(* IEC 61131-3 sources: plc_simulator/services/codesys/POUs (part 10) *)

(* ---- TSK_FB_Analyze.st ---- *)
(* ============================================================
   TSK_FB_Analyze — Conflict analysis for task list
   ============================================================
   Ported from transporterTaskScheduler.js analyzeTaskConflicts()

   Three conflict checks, each stops at first hit:

   1. TASK_SEQUENCE: per-transporter queue order (preserves SWAP).
      Does the transporter have time to travel from prev.sink
      to next.lift?

   2. TRANSPORTER_COLLISION: different transporters — do their
      X-ranges and time-ranges overlap?

   3. CROSS_TRANSPORTER_HANDOFF: same batch, consecutive stages
      on different transporters — does the receiving transporter
      have time to reach the handoff station?

   NOTE: TASK_SEQUENCE iterates g_task[ti].Queue[] directly
   (not a merged sorted list) so SWAP ordering is preserved.

   Outputs:
     o_has_conflict — TRUE if conflict found
     o_conf_unit, o_conf_stage — which task is blocked
     o_blocked_unit, o_blocked_stage — which task blocks it
     o_deficit — how many seconds short
     o_conf_type — 1=TASK_SEQUENCE, 2=COLLISION, 3=HANDOFF
     checked_count — total tasks inspected
   ============================================================ *)

FUNCTION_BLOCK TSK_FB_Analyze
VAR_EXTERNAL CONSTANT
    MAX_Transporters    : INT;
    MAX_Units           : INT;
    MIN_StationIndex : INT;
    MAX_StationIndex   : INT;
END_VAR

VAR_EXTERNAL
  g_task    : ARRAY[1..MAX_Transporters] OF UDT_JC_TskQueueType;
  g_station : ARRAY[MIN_StationIndex..MAX_StationIndex] OF UDT_StationType;
  g_move    : ARRAY[1..MAX_Transporters] OF UDT_JC_MoveTimesType;
END_VAR
VAR_OUTPUT
  o_has_conflict  : BOOL;
  o_conf_type     : INT;     (* 1=TASK_SEQUENCE, 2=COLLISION, 3=HANDOFF *)
  o_conf_unit     : INT;     (* conflict task: unit *)
  o_conf_stage    : INT;     (* conflict task: stage *)
  o_conf_trans    : INT;     (* conflict task: transporter *)
  o_blocked_unit  : INT;     (* blocking task: unit *)
  o_blocked_stage : INT;     (* blocking task: stage *)
  o_deficit       : REAL;    (* seconds short *)
  checked_count   : INT;     (* tasks checked before conflict *)
END_VAR
VAR
  (* Loop variables *)
  ti       : INT;    (* transporter outer *)
  tj       : INT;    (* transporter inner *)
  qi       : INT;    (* queue index outer *)
  qj       : INT;    (* queue index inner *)
  (* TASK_SEQUENCE *)
  prev_sink : INT;
  next_lift : INT;
  travel_s  : REAL;
  gap_s     : REAL;
  deficit_s : REAL;
  (* TRANSPORTER_COLLISION: X range per task *)
  lift_x   : REAL;
  sink_x   : REAL;
  x1_min   : REAL;
  x1_max   : REAL;
  x2_min   : REAL;
  x2_max   : REAL;
  xo_start : REAL;
  xo_end   : REAL;
  to_start : LINT;
  to_end   : LINT;
  l_idx    : INT;
  s_idx    : INT;
  lift_x2  : REAL;
  sink_x2  : REAL;
  l_idx2   : INT;
  s_idx2   : INT;
  (* CROSS_TRANSPORTER_HANDOFF *)
  cur_unit    : INT;
  cur_stage   : INT;
  found_next  : BOOL;
  recv_prev_end  : LINT;
  recv_prev_sink : INT;
  has_recv_prev  : BOOL;
  rk       : INT;     (* receiver prev search *)
  recv_prev_unit : INT;    (* saved receiver prev task unit *)
  recv_prev_stg  : INT;    (* saved receiver prev task stage *)
  recv_travel    : REAL;
  recv_earliest  : LINT;
  handoff_deficit : REAL;
  (* Counter *)
  total_tasks : INT;
  DEFICIT_TOL : REAL := 1.0;
  tmp_move    : UDT_JC_MoveTimesType;  (* MATIEC cannot index arrays in FUNCTION args *)
END_VAR

o_has_conflict := FALSE;
o_conf_type    := 0;
o_deficit      := 0.0;
checked_count  := 0;

(* Count total tasks *)
total_tasks := 0;
FOR ti := 1 TO MAX_Transporters DO
  total_tasks := total_tasks + g_task[ti].Count;
END_FOR;
IF total_tasks = 0 THEN RETURN; END_IF;

(* ══════════════════════════════════════════════════════════════════════ *)
(* CHECK 1: TASK_SEQUENCE — per-transporter queue order (SWAP-safe)    *)
(* Iterates g_task[ti].Queue[] in queue order, NOT sorted by time.     *)
(* ══════════════════════════════════════════════════════════════════════ *)
FOR ti := 1 TO MAX_Transporters DO
  FOR qi := 1 TO g_task[ti].Count - 1 DO
    IF g_task[ti].Queue[qi].Unit > 0 AND g_task[ti].Queue[qi + 1].Unit > 0 THEN

      prev_sink := g_task[ti].Queue[qi].SinkStationTarget;
      next_lift := g_task[ti].Queue[qi + 1].LiftStationTarget;

      tmp_move := g_move[ti];
      travel_s := STC_CalcHorizontalTravel(i_from_stn := prev_sink, i_to_stn := next_lift, i_move := tmp_move);

      gap_s := LINT_TO_REAL(
        g_task[ti].Queue[qi + 1].StartTime - g_task[ti].Queue[qi].FinishTime
      );
      deficit_s := travel_s - gap_s;

      IF deficit_s > DEFICIT_TOL THEN
        o_has_conflict  := TRUE;
        o_conf_type     := 1;  (* TASK_SEQUENCE *)
        o_conf_unit     := g_task[ti].Queue[qi + 1].Unit;
        o_conf_stage    := g_task[ti].Queue[qi + 1].Stage;
        o_conf_trans    := ti;
        o_blocked_unit  := g_task[ti].Queue[qi].Unit;
        o_blocked_stage := g_task[ti].Queue[qi].Stage;
        o_deficit       := deficit_s;
        checked_count   := total_tasks;
        RETURN;
      END_IF;

    END_IF;
  END_FOR;
END_FOR;

(* ══════════════════════════════════════════════════════════════════════ *)
(* CHECK 2: CROSS_TRANSPORTER_HANDOFF                                  *)
(* Same batch, consecutive stages on different transporters.           *)
(* Does the receiving transporter have time to reach handoff station?  *)
(*                                                                      *)
(* JS checks HANDOFF before COLLISION (per-task loop order).           *)
(* Conflict targets the DELIVERING task (current transporter);         *)
(* resolver will delay the preceding stage so the batch waits longer   *)
(* on the delivering transporter's side.                               *)
(* ══════════════════════════════════════════════════════════════════════ *)
FOR ti := 1 TO MAX_Transporters DO
  FOR qi := 1 TO g_task[ti].Count DO
    cur_unit  := g_task[ti].Queue[qi].Unit;
    cur_stage := g_task[ti].Queue[qi].Stage;
    IF cur_unit > 0 THEN

      (* Find next stage of same batch in a different transporter *)
      found_next := FALSE;
      FOR tj := 1 TO MAX_Transporters DO
        IF tj <> ti AND NOT found_next THEN
          FOR qj := 1 TO g_task[tj].Count DO
            IF NOT found_next THEN
              IF g_task[tj].Queue[qj].Unit = cur_unit
                 AND g_task[tj].Queue[qj].Stage = cur_stage + 1 THEN
                found_next := TRUE;

                (* Found handoff pair: ti delivers to sink, tj picks up *)
                (* Find receiver's (tj) previous task — latest finish before next task start *)
                has_recv_prev := FALSE;
                recv_prev_end  := 0;
                recv_prev_sink := 0;
                recv_prev_unit := 0;
                recv_prev_stg  := 0;
                FOR rk := 1 TO g_task[tj].Count DO
                  IF rk <> qj THEN
                    IF g_task[tj].Queue[rk].FinishTime <= g_task[tj].Queue[qj].StartTime THEN
                      IF NOT has_recv_prev OR g_task[tj].Queue[rk].FinishTime > recv_prev_end THEN
                        has_recv_prev := TRUE;
                        recv_prev_end  := g_task[tj].Queue[rk].FinishTime;
                        recv_prev_sink := g_task[tj].Queue[rk].SinkStationTarget;
                        recv_prev_unit := g_task[tj].Queue[rk].Unit;
                        recv_prev_stg  := g_task[tj].Queue[rk].Stage;
                      END_IF;
                    END_IF;
                  END_IF;
                END_FOR;

                IF has_recv_prev THEN
                  (* Travel from receiver's prev sink to handoff station (= ti's current sink) *)
                  recv_travel := STC_CalcHorizontalTravel(
                    i_from_stn := recv_prev_sink,
                    i_to_stn   := g_task[ti].Queue[qi].SinkStationTarget,
                    i_move     := g_move[tj]
                  );
                  recv_earliest := recv_prev_end + REAL_TO_LINT(recv_travel);
                  handoff_deficit := LINT_TO_REAL(
                    recv_earliest - g_task[ti].Queue[qi].FinishTime
                  );

                  IF handoff_deficit > DEFICIT_TOL THEN
                    o_has_conflict  := TRUE;
                    o_conf_type     := 3;  (* CROSS_TRANSPORTER_HANDOFF *)
                    (* Conflict on delivering task *)
                    o_conf_unit     := g_task[ti].Queue[qi].Unit;
                    o_conf_stage    := g_task[ti].Queue[qi].Stage;
                    o_conf_trans    := ti;
                    (* Blocked by receiver's previous task *)
                    o_blocked_unit  := recv_prev_unit;
                    o_blocked_stage := recv_prev_stg;
                    o_deficit       := handoff_deficit;
                    checked_count   := total_tasks;
                    RETURN;
                  END_IF;
                END_IF;
                (* If no recv prev task, receiver is idle → no handoff conflict *)

              END_IF;
            END_IF;
          END_FOR;
        END_IF;
      END_FOR;

    END_IF;
  END_FOR;
END_FOR;

(* ══════════════════════════════════════════════════════════════════════ *)
(* CHECK 3: TRANSPORTER_COLLISION — X+time overlap, different trans.   *)
(* Compares every task pair across different transporters.              *)
(* JS: conf = later task (timeline), blocked = earlier task.           *)
(* ══════════════════════════════════════════════════════════════════════ *)
FOR ti := 1 TO MAX_Transporters DO
  FOR qi := 1 TO g_task[ti].Count DO
    IF g_task[ti].Queue[qi].Unit > 0 THEN

      (* X range for task A *)
      l_idx := g_task[ti].Queue[qi].LiftStationTarget - 100;
      s_idx := g_task[ti].Queue[qi].SinkStationTarget - 100;
      IF l_idx >= 1 AND l_idx <= 30 THEN
        lift_x := DINT_TO_REAL(g_station[g_task[ti].Queue[qi].LiftStationTarget].XPosition);
      ELSE
        lift_x := 0.0;
      END_IF;
      IF s_idx >= 1 AND s_idx <= 30 THEN
        sink_x := DINT_TO_REAL(g_station[g_task[ti].Queue[qi].SinkStationTarget].XPosition);
      ELSE
        sink_x := 0.0;
      END_IF;
      IF lift_x < sink_x THEN
        x1_min := lift_x;
        x1_max := sink_x;
      ELSE
        x1_min := sink_x;
        x1_max := lift_x;
      END_IF;

      FOR tj := ti + 1 TO MAX_Transporters DO
        FOR qj := 1 TO g_task[tj].Count DO
          IF g_task[tj].Queue[qj].Unit > 0 THEN

            (* X range for task B *)
            l_idx2 := g_task[tj].Queue[qj].LiftStationTarget - 100;
            s_idx2 := g_task[tj].Queue[qj].SinkStationTarget - 100;
            IF l_idx2 >= 1 AND l_idx2 <= 30 THEN
              lift_x2 := DINT_TO_REAL(g_station[g_task[tj].Queue[qj].LiftStationTarget].XPosition);
            ELSE
              lift_x2 := 0.0;
            END_IF;
            IF s_idx2 >= 1 AND s_idx2 <= 30 THEN
              sink_x2 := DINT_TO_REAL(g_station[g_task[tj].Queue[qj].SinkStationTarget].XPosition);
            ELSE
              sink_x2 := 0.0;
            END_IF;
            IF lift_x2 < sink_x2 THEN
              x2_min := lift_x2;
              x2_max := sink_x2;
            ELSE
              x2_min := sink_x2;
              x2_max := lift_x2;
            END_IF;

            (* X overlap *)
            xo_start := x1_min;
            IF x2_min > xo_start THEN xo_start := x2_min; END_IF;
            xo_end := x1_max;
            IF x2_max < xo_end THEN xo_end := x2_max; END_IF;

            IF xo_start < xo_end THEN
              (* Time overlap *)
              to_start := g_task[ti].Queue[qi].StartTime;
              IF g_task[tj].Queue[qj].StartTime > to_start THEN
                to_start := g_task[tj].Queue[qj].StartTime;
              END_IF;
              to_end := g_task[ti].Queue[qi].FinishTime;
              IF g_task[tj].Queue[qj].FinishTime < to_end THEN
                to_end := g_task[tj].Queue[qj].FinishTime;
              END_IF;

              IF to_start < to_end THEN
                deficit_s := LINT_TO_REAL(to_end - to_start) + 2.0;
                o_has_conflict  := TRUE;
                o_conf_type     := 2;  (* TRANSPORTER_COLLISION *)
                (* Assign conf = later task (timeline), blocked = earlier task — matches JS *)
                IF g_task[ti].Queue[qi].StartTime <= g_task[tj].Queue[qj].StartTime THEN
                  o_conf_unit     := g_task[tj].Queue[qj].Unit;
                  o_conf_stage    := g_task[tj].Queue[qj].Stage;
                  o_conf_trans    := tj;
                  o_blocked_unit  := g_task[ti].Queue[qi].Unit;
                  o_blocked_stage := g_task[ti].Queue[qi].Stage;
                ELSE
                  o_conf_unit     := g_task[ti].Queue[qi].Unit;
                  o_conf_stage    := g_task[ti].Queue[qi].Stage;
                  o_conf_trans    := ti;
                  o_blocked_unit  := g_task[tj].Queue[qj].Unit;
                  o_blocked_stage := g_task[tj].Queue[qj].Stage;
                END_IF;
                o_deficit       := deficit_s;
                checked_count   := total_tasks;
                RETURN;
              END_IF;
            END_IF;

          END_IF;
        END_FOR;
      END_FOR;

    END_IF;
  END_FOR;
END_FOR;

(* No conflict found *)
checked_count := total_tasks;

END_FUNCTION_BLOCK

(* ---- TSK_FB_CalcSchedule.st ---- *)
(* ============================================================
   TSK_FB_CalcSchedule — Calculate batch schedule for one unit
   ============================================================
   Ported from transporterTaskScheduler.js calculateBatchSchedule()

   Calculates schedule timeline for one unit/batch:
   - Reads treatment program stages
   - Calculates transfer times from g_move
   - Writes entry/exit times to g_schedule[unit]

   Parallel stations: picks first available (stations[1] default).
   Transfer time: lift + travel + sink from g_move precomputed table.

   Called once per batch per scheduler cycle.
   ============================================================ *)

FUNCTION_BLOCK TSK_FB_CalcSchedule
VAR_INPUT
  i_unit     : INT;     (* unit index 1..10 *)
  i_trans    : INT;     (* transporter index 1..3 for move times *)
  i_time_s   : LINT;    (* current absolute time (s), unix seconds *)
END_VAR
VAR_EXTERNAL CONSTANT
    MIN_StationIndex : INT;
    MAX_StationIndex   : INT;
    MAX_Units           : INT;
    MAX_Transporters    : INT;
END_VAR
VAR_EXTERNAL
  g_batch  : ARRAY[1..MAX_Units] OF UDT_BatchType;
  g_program : ARRAY[1..MAX_Units] OF UDT_TreatmentProgramType;
  g_unit    : ARRAY[1..MAX_Units] OF UDT_UnitType;
  g_station : ARRAY[MIN_StationIndex..MAX_StationIndex] OF UDT_StationType;
  g_station_loc : ARRAY[1..MAX_StationIndex] OF UDT_UnitLocation;
  g_schedule : ARRAY[1..MAX_Units] OF UDT_JC_TskScheduleType;
  g_station_count : INT;
  g_move    : ARRAY[1..MAX_Transporters] OF UDT_JC_MoveTimesType;
  g_cfg     : ARRAY[1..MAX_Transporters] OF UDT_TransporterType;
  g_transporter : ARRAY[1..MAX_Transporters] OF UDT_TransporterStatusType;
END_VAR
VAR
  stg         : INT;      (* loop: stage index *)
  stn_num    : INT;      (* target station number *)
  prev_stn   : INT;      (* previous station number *)
  cur_stage  : INT;      (* batch current stage *)
  location   : INT;      (* unit location *)
  start_st   : INT;      (* first stage to calculate *)
  entry_t    : LINT;     (* entry time for stage, absolute *)
  exit_t     : LINT;     (* exit time for stage, absolute *)
  xfer_t     : REAL;     (* transfer time *)
  calc_s     : REAL;     (* calc_time in seconds *)
  min_s      : REAL;     (* min_time in seconds *)
  max_s      : REAL;     (* max_time in seconds *)
  is_on_stn  : BOOL;     (* TRUE if unit is on a station *)
  is_first   : BOOL;     (* TRUE for first stage in loop *)
  remain_s   : REAL;     (* remaining time on current station *)
  elapsed_s  : REAL;     (* elapsed time on current station *)
  out_count  : INT;      (* output stage counter *)
  p          : INT;      (* parallel station loop index *)
  chosen_stn : INT;      (* chosen parallel station *)
  tmp_move   : UDT_JC_MoveTimesType;  (* MATIEC cannot index arrays in FUNCTION args *)
  (* ── Parallel station selection (schedule-aware + idle-since) ── *)
  cand_arr         : ARRAY[1..5] OF INT;
  cand_cnt         : INT;
  sched_occupied   : ARRAY[1..5] OF BOOL;
  phys_occupied    : ARRAY[1..5] OF BOOL;
  best_change_time : LINT;
  my_entry         : LINT;
  my_exit          : LINT;
  ov_start         : LINT;
  ov_end           : LINT;
  uj               : INT;
  sj               : INT;
  saved_entry_t    : LINT;  (* previous cycle's first-stage EntryTime for on-transporter clamp *)
END_VAR

(* -- Validate inputs -- *)
IF i_unit < 1 OR i_unit > MAX_Units THEN RETURN; END_IF;
IF i_trans < 1 OR i_trans > MAX_Transporters THEN RETURN; END_IF;

(* -- Read batch and unit data -- *)
cur_stage := g_batch[i_unit].CurStage;
location  := g_unit[i_unit].location;
is_on_stn := location >= 100;
out_count := 0;

(* -- Save previous first-stage entry time before clearing -- *)
(* When unit is on transporter, we preserve the previously calculated
   entry time as long as it is still in the future (= transporter on schedule).
   If it has passed, we clamp to now (= transporter is late). *)
saved_entry_t := 0;
IF NOT is_on_stn AND g_schedule[i_unit].StageCount > 0 THEN
  saved_entry_t := g_schedule[i_unit].Stages[1].EntryTime;
END_IF;

(* -- Clear old schedule -- *)
FOR stg := 1 TO 30 DO
  g_schedule[i_unit].Stages[stg].station := 0;
  g_schedule[i_unit].Stages[stg].ProgramStage := 0;
  g_schedule[i_unit].Stages[stg].EntryTime := 0;
  g_schedule[i_unit].Stages[stg].ExitTime := 0;
  g_schedule[i_unit].Stages[stg].MinTime := 0;
  g_schedule[i_unit].Stages[stg].CalcTime := 0;
  g_schedule[i_unit].Stages[stg].MaxTime := 0;
  g_schedule[i_unit].Stages[stg].TransferTime := 0;
END_FOR;

(* -- Determine start stage -- *)
(* Waiting batch (state = NOT_PROCESSED): treat as stage 0 *)
IF g_batch[i_unit].State = 0 THEN
  cur_stage := 0;
END_IF;

(* If on transporter, start from next stage; if on station, from current *)
IF is_on_stn THEN
  start_st := cur_stage;
ELSE
  start_st := cur_stage + 1;
END_IF;

(* Force minimum stage 1 *)
IF start_st < 1 THEN
  start_st := 1;
END_IF;

(* -- Previous station (where transfer starts from) -- *)
IF is_on_stn THEN
  prev_stn := location;
ELSIF cur_stage >= 1 AND cur_stage <= 30 THEN
  (* On transporter: use previous stage station *)
  prev_stn := g_program[i_unit].Steps[cur_stage].Stations[0];
ELSE
  prev_stn := 0;
END_IF;

(* -- prevExitTime: when next stage can begin -- *)
exit_t := i_time_s;

is_first := TRUE;

(* -- Prepend current location when unit needs pre-positioning -- *)
(* If unit is on a station that is NOT the first treatment station,
   insert it as schedule entry 0 (0 treatment time) so that
   CreateTasks generates a move-to-first-station task. *)
IF is_on_stn AND start_st >= 1 THEN
  stn_num := 0;
  FOR p := 0 TO 4 DO
    IF g_program[i_unit].Steps[start_st].Stations[p] = location THEN
      stn_num := location;  (* flag: already on first treatment station *)
    END_IF;
  END_FOR;
  IF stn_num = 0 THEN
    out_count := out_count + 1;
    g_schedule[i_unit].Stages[out_count].station       := location;
    g_schedule[i_unit].Stages[out_count].ProgramStage := 0;  (* pre-position entry, not a program stage *)
    g_schedule[i_unit].Stages[out_count].EntryTime    := exit_t;
    g_schedule[i_unit].Stages[out_count].TransferTime := 0;

    (* ── Stage 0 times from batch data — JS: stage0 prepend uses batch.calc/min/max ──
       CurStage=0 means just activated: use batch CalTime (= remaining wait time)
       Otherwise (mid-process repositioning): zero duration *)
    IF g_batch[i_unit].CurStage = 0 AND g_batch[i_unit].CalTime > 0 THEN
      (* JS: remainingSec = max(1, calcTimeS - elapsed) *)
      IF g_batch[i_unit].StartTime > 0 AND g_batch[i_unit].StartTime < i_time_s THEN
        elapsed_s := LINT_TO_REAL(i_time_s - g_batch[i_unit].StartTime);
      ELSE
        elapsed_s := 0.0;
      END_IF;
      remain_s := DINT_TO_REAL(g_batch[i_unit].CalTime) - elapsed_s;
      IF remain_s < 1.0 THEN remain_s := 1.0; END_IF;
      exit_t := i_time_s + REAL_TO_LINT(remain_s);
      g_schedule[i_unit].Stages[out_count].ExitTime  := exit_t;
      g_schedule[i_unit].Stages[out_count].CalcTime  := REAL_TO_DINT(remain_s);
      g_schedule[i_unit].Stages[out_count].MinTime   := g_batch[i_unit].MinTime;
      g_schedule[i_unit].Stages[out_count].MaxTime   := g_batch[i_unit].MaxTime;
    ELSE
      g_schedule[i_unit].Stages[out_count].ExitTime  := exit_t;
      g_schedule[i_unit].Stages[out_count].CalcTime  := 0;
      g_schedule[i_unit].Stages[out_count].MinTime   := 0;
      g_schedule[i_unit].Stages[out_count].MaxTime   := 0;
    END_IF;

    is_first := FALSE;
  END_IF;
END_IF;

(* ============================================================
   MAIN LOOP: Calculate schedule for each program stage
   ============================================================ *)
FOR stg := start_st TO g_program[i_unit].StepCount DO

  (* Check if stage has valid stations — parallel selection *)
  cand_cnt := 0;
  FOR p := 0 TO 4 DO
    IF g_program[i_unit].Steps[stg].Stations[p] > 0 THEN
      cand_cnt := cand_cnt + 1;
      cand_arr[cand_cnt] := g_program[i_unit].Steps[stg].Stations[p];
      sched_occupied[cand_cnt] := FALSE;
      phys_occupied[cand_cnt] := FALSE;
    END_IF;
  END_FOR;

  (* No station means end of program *)
  IF cand_cnt = 0 THEN
    EXIT;
  END_IF;

  IF cand_cnt = 1 THEN
    chosen_stn := cand_arr[1];
  ELSE
    (* Read treatment times early — needed for time window estimate *)
    calc_s := DINT_TO_REAL(g_program[i_unit].Steps[stg].CalTime);

    (* Estimate this stage's time window *)
    tmp_move := g_move[i_trans];
    xfer_t := STC_CalcTransferTime(
      i_from_stn            := prev_stn,
      i_to_stn              := cand_arr[1],
      i_move                := tmp_move,
      i_from_dropping_x10   := g_station[prev_stn].DrippingTime,
      i_to_device_delay_x10 := g_station[cand_arr[1]].DeviceDelay,
      i_drip_tray_delay_x10 := g_cfg[i_trans].DripTrayDelay
    );
    my_entry := exit_t + REAL_TO_LINT(xfer_t);
    my_exit  := my_entry + REAL_TO_LINT(calc_s);

    (* Check schedule overlap + physical occupation for each candidate *)
    FOR p := 1 TO cand_cnt DO
      FOR uj := 1 TO MAX_Units DO
        IF uj <> i_unit AND g_schedule[uj].StageCount > 0 THEN
          FOR sj := 1 TO g_schedule[uj].StageCount DO
            IF g_schedule[uj].Stages[sj].station = cand_arr[p] THEN
              ov_start := my_entry;
              IF g_schedule[uj].Stages[sj].EntryTime > ov_start THEN
                ov_start := g_schedule[uj].Stages[sj].EntryTime;
              END_IF;
              ov_end := my_exit;
              IF g_schedule[uj].Stages[sj].ExitTime < ov_end THEN
                ov_end := g_schedule[uj].Stages[sj].ExitTime;
              END_IF;
              IF ov_end > ov_start THEN
                sched_occupied[p] := TRUE;
              END_IF;
            END_IF;
          END_FOR;
        END_IF;
      END_FOR;

      (* Physical occupation *)
      FOR uj := 1 TO MAX_Units DO
        IF g_unit[uj].location = cand_arr[p] AND g_unit[uj].Status = 1 THEN
          phys_occupied[p] := TRUE;
        END_IF;
      END_FOR;
    END_FOR;

    (* Select best free station: longest idle = smallest change_time *)
    chosen_stn := 0;
    best_change_time := LINT#9999999999;
    FOR p := 1 TO cand_cnt DO
      IF NOT sched_occupied[p] AND NOT phys_occupied[p] THEN
        IF cand_arr[p] >= MIN_StationIndex AND cand_arr[p] <= MAX_StationIndex THEN
          IF g_station_loc[cand_arr[p]].ChangeTime < best_change_time THEN
            best_change_time := g_station_loc[cand_arr[p]].ChangeTime;
            chosen_stn := cand_arr[p];
          END_IF;
        END_IF;
      END_IF;
    END_FOR;

    (* Fallback: schedule-free only *)
    IF chosen_stn = 0 THEN
      FOR p := 1 TO cand_cnt DO
        IF NOT sched_occupied[p] AND chosen_stn = 0 THEN
          chosen_stn := cand_arr[p];
        END_IF;
      END_FOR;
    END_IF;

    (* Ultimate fallback: first candidate *)
    IF chosen_stn = 0 THEN
      chosen_stn := cand_arr[1];
    END_IF;
  END_IF;

  stn_num := chosen_stn;

  (* Read treatment times from program *)
  calc_s := DINT_TO_REAL(g_program[i_unit].Steps[stg].CalTime);
  min_s  := DINT_TO_REAL(g_program[i_unit].Steps[stg].MinTime);
  max_s  := DINT_TO_REAL(g_program[i_unit].Steps[stg].MaxTime);

  (* -- Calculate transfer time from prev_stn to stn_num -- *)
  (* Cross-transfer check: if prev_stn has Crosstransport and different Y line
     → use ChangeStation as effective source for transfer time calc
     JS: calculateTransferTimeWithCrossCheck *)
  tmp_move := g_move[i_trans];
  (* ST does NOT short-circuit AND — bounds must be checked in separate IF
     before any g_station[prev_stn] or g_station[stn_num] access *)
  IF prev_stn >= MIN_StationIndex AND prev_stn <= MAX_StationIndex
     AND stn_num >= MIN_StationIndex AND stn_num <= MAX_StationIndex THEN
    IF g_station[prev_stn].Crosstransport > 0
       AND g_station[prev_stn].ChangeStation > 0
       AND g_station[prev_stn].YPosition <> g_station[stn_num].YPosition THEN
      (* Cross-transfer: belt time + transfer from ChangeStation to sink *)
      xfer_t := INT_TO_REAL(g_station[prev_stn].CrossTransportTime)
              + STC_CalcTransferTime(
                  i_from_stn            := g_station[prev_stn].ChangeStation,
                  i_to_stn              := stn_num,
                  i_move                := tmp_move,
                  i_from_dropping_x10   := g_station[g_station[prev_stn].ChangeStation].DrippingTime,
                  i_to_device_delay_x10 := g_station[stn_num].DeviceDelay,
                  i_drip_tray_delay_x10 := g_cfg[i_trans].DripTrayDelay
                );
    ELSE
      xfer_t := STC_CalcTransferTime(
        i_from_stn            := prev_stn,
        i_to_stn              := stn_num,
        i_move                := tmp_move,
        i_from_dropping_x10   := g_station[prev_stn].DrippingTime,
        i_to_device_delay_x10 := g_station[stn_num].DeviceDelay,
        i_drip_tray_delay_x10 := g_cfg[i_trans].DripTrayDelay
      );
    END_IF;
  ELSE
    (* Out-of-range station index — use safe fallback *)
    xfer_t := 60.0;
  END_IF;

  (* -- Calculate entry and exit times -- *)
  IF is_first AND is_on_stn AND stg = cur_stage THEN
    (* Batch is currently at this station *)
    entry_t := i_time_s;
    (* Remaining time: use g_batch[].CalTime (resolver-modified)
       JS: remainingTimeS = max(1, batch.calc_time_s - elapsed) *)
    IF g_batch[i_unit].StartTime > 0 THEN
      elapsed_s := LINT_TO_REAL(i_time_s - g_batch[i_unit].StartTime);
    ELSE
      elapsed_s := 0.0;
    END_IF;
    remain_s := DINT_TO_REAL(g_batch[i_unit].CalTime) - elapsed_s;
    IF remain_s < 1.0 THEN remain_s := 1.0; END_IF;
    exit_t := i_time_s + REAL_TO_LINT(remain_s);
  ELSIF is_first AND NOT is_on_stn THEN
    (* Batch is on transporter — use saved entry time from previous cycle.
       If transporter is on schedule (saved > now), keep it stable.
       If transporter is late (saved <= now), clamp to now. *)
    IF saved_entry_t > i_time_s THEN
      entry_t := saved_entry_t;  (* on schedule — keep stable *)
    ELSE
      entry_t := i_time_s;       (* late or first cycle — clamp to now *)
    END_IF;
    exit_t  := entry_t + REAL_TO_LINT(calc_s);
  ELSE
    (* Normal stage: entry = prev exit + transfer *)
    entry_t := exit_t + REAL_TO_LINT(xfer_t);
    exit_t  := entry_t + REAL_TO_LINT(calc_s);
  END_IF;

  (* -- Write to schedule -- *)
  out_count := out_count + 1;
  IF out_count <= 30 THEN
    g_schedule[i_unit].Stages[out_count].station       := stn_num;
    g_schedule[i_unit].Stages[out_count].ProgramStage := stg;  (* program stage number (1..N) *)
    g_schedule[i_unit].Stages[out_count].EntryTime    := entry_t;
    g_schedule[i_unit].Stages[out_count].ExitTime     := exit_t;
    g_schedule[i_unit].Stages[out_count].MinTime      := REAL_TO_DINT(min_s);
    g_schedule[i_unit].Stages[out_count].CalcTime     := REAL_TO_DINT(calc_s);
    g_schedule[i_unit].Stages[out_count].MaxTime      := REAL_TO_DINT(max_s);
    g_schedule[i_unit].Stages[out_count].TransferTime := REAL_TO_DINT(xfer_t);
  END_IF;

  (* -- Update for next iteration -- *)
  prev_stn := stn_num;
  is_first := FALSE;

END_FOR;

g_schedule[i_unit].StageCount := out_count;

END_FUNCTION_BLOCK

(* ---- TSK_FB_CreateTasks.st ---- *)
(* ============================================================
   TSK_FB_CreateTasks — Build task list from schedule
   ============================================================
   Ported from transporterTaskScheduler.js createTaskListFromSchedule()

   For each consecutive stage pair in g_schedule[unit]:
     - Lift station = current stage station
     - Sink station = next stage station
     - Assigns transporter from task_area match in g_cfg
     - Skips already completed stages (stage < batch.CurStage)
   Appends tasks to g_task[transporter].Queue.

   Called once per batch per scheduler cycle.
   ============================================================ *)

FUNCTION_BLOCK TSK_FB_CreateTasks
VAR_INPUT
  i_unit : INT;   (* unit index 1..10 *)
END_VAR
VAR_EXTERNAL CONSTANT
    MAX_Transporters : INT;
    MAX_Units        : INT;
    MAX_TASK_QUEUE   : INT;
    MIN_StationIndex : INT;
    MAX_StationIndex : INT;
END_VAR

VAR_EXTERNAL
  g_batch  : ARRAY[1..MAX_Units] OF UDT_BatchType;
  g_schedule : ARRAY[1..MAX_Units] OF UDT_JC_TskScheduleType;
  g_task    : ARRAY[1..MAX_Transporters] OF UDT_JC_TskQueueType;
  g_cfg    : ARRAY[1..MAX_Transporters] OF UDT_TransporterType;
  g_station : ARRAY[MIN_StationIndex..MAX_StationIndex] OF UDT_StationType;
END_VAR
VAR
  si         : INT;     (* schedule stage index *)
  sc         : INT;     (* stage count *)
  lift_stn   : INT;     (* lift station *)
  sink_stn   : INT;     (* sink station *)
  tid        : INT;     (* transporter id found *)
  qi         : INT;     (* queue write index *)
  fb_find    : STC_FindTransporter;  (* transporter lookup *)
  (* Cross-transfer detection — JS: isCrossTransporterOp + findCrossTransporterEndStation *)
  eff_lift_stn : INT;   (* effective lift station after cross-transfer check *)
END_VAR

IF i_unit < 1 OR i_unit > MAX_Units THEN RETURN; END_IF;

sc := g_schedule[i_unit].StageCount;
IF sc < 2 THEN RETURN; END_IF;

(* CalcSchedule already builds a schedule starting from the batch's
   current stage (and prepends the unit's current location when needed).
   No skip logic needed here — every consecutive pair is a valid task. *)

(* Loop through consecutive stage pairs *)
FOR si := 1 TO sc - 1 DO
  lift_stn := g_schedule[i_unit].Stages[si].station;
  sink_stn := g_schedule[i_unit].Stages[si + 1].station;

  IF lift_stn > 0 AND sink_stn > 0 THEN
    (* -- Cross-transfer detection -- *)
    (* JS: if station.operation === 10 && lift.y_position !== sink.y_position
       → use ChangeStation as effective lift (belt other end, same line as sink) *)
    eff_lift_stn := lift_stn;
    IF lift_stn >= MIN_StationIndex AND lift_stn <= MAX_StationIndex
       AND sink_stn >= MIN_StationIndex AND sink_stn <= MAX_StationIndex THEN
      IF g_station[lift_stn].Crosstransport > 0
         AND g_station[lift_stn].ChangeStation > 0
         AND g_station[lift_stn].YPosition <> g_station[sink_stn].YPosition THEN
        eff_lift_stn := g_station[lift_stn].ChangeStation;
      END_IF;
    END_IF;

    (* -- Find transporter via task_area matching (with scoring) -- *)
    fb_find(i_lift_stn := eff_lift_stn, i_sink_stn := sink_stn);
    tid := fb_find.o_trans;

    (* -- Append task to transporter queue -- *)
    IF tid >= 1 AND tid <= 3 THEN
      qi := g_task[tid].Count + 1;
      IF qi <= MAX_TASK_QUEUE THEN
        g_task[tid].Queue[qi].Unit         := i_unit;
        g_task[tid].Queue[qi].Stage        := g_schedule[i_unit].Stages[si].ProgramStage;  (* program stage — direct index to g_program.Steps[] *)
        g_task[tid].Queue[qi].LiftStationTarget := eff_lift_stn;
        g_task[tid].Queue[qi].SinkStationTarget := sink_stn;
        g_task[tid].Queue[qi].StartTime   := g_schedule[i_unit].Stages[si].ExitTime;
        g_task[tid].Queue[qi].FinishTime  := g_schedule[i_unit].Stages[si + 1].EntryTime;
        g_task[tid].Queue[qi].CalcTime    := g_schedule[i_unit].Stages[si].CalcTime;
        g_task[tid].Queue[qi].MinTime     := g_schedule[i_unit].Stages[si].MinTime;
        g_task[tid].Queue[qi].MaxTime     := g_schedule[i_unit].Stages[si].MaxTime;
        g_task[tid].Count := qi;
      END_IF;
    END_IF;
  END_IF;
END_FOR;

END_FUNCTION_BLOCK

(* ---- TSK_FB_NoTreatment.st ---- *)
(* ============================================================
   TSK_FB_NoTreatment — Create no-treatment transfer tasks
   ============================================================
   Scans units that have a target (TO_LOADING, TO_UNLOAD,
   TO_BUFFER, TO_AVOID, etc.) and creates transfer tasks using
   the g_ntt destination table (per target, per transporter).

   Destination lookup:
     1. Search primary stations (g_ntt[trans].Target[tgt].Stations)
     2. If all occupied → search fallback stations
     3. First free station wins

   Conditions for creating a task:
     - Unit has target <> TO_NONE
     - TO_PROCESS handled only when batch state = NOT_PROCESSED
       (routes to loaded-buffer via NTT index 7)
     - Unit is on a station (location >= 100)
     - Covering transporter is idle (phase = 0, active)
     - A free destination station exists in g_ntt
     - Destination station MUST be actually free (no unit present)
     - No overlap conflict with OTHER transporters that share the
       destination area (mirrors JS _hasOverlapConflict):
       * If another transporter also covers dest_stn and is actively
         moving (Phase 1-4) with its task in the shared zone → skip
       * If another transporter has queued tasks that overlap in time
         AND operate in cov_t's task area → skip
   ============================================================ *)

FUNCTION_BLOCK TSK_FB_NoTreatment
VAR_INPUT
  i_time_s : LINT;   (* current absolute time (s), unix seconds *)
END_VAR
VAR_EXTERNAL CONSTANT
    MAX_Transporters    : INT;
    MAX_STATIONS_PER_STEP       : INT;
    MIN_StationIndex : INT;
    MAX_StationIndex   : INT;
    MAX_Units           : INT;
    MAX_TASK_QUEUE      : INT;
END_VAR

VAR_EXTERNAL
  g_unit        : ARRAY[1..MAX_Units] OF UDT_UnitType;
  g_batch       : ARRAY[1..MAX_Units] OF UDT_BatchType;
  g_ntt         : ARRAY[1..MAX_Transporters] OF UDT_JC_NttTransporterType;
  g_transporter : ARRAY[1..MAX_Transporters] OF UDT_TransporterStatusType;
  g_station     : ARRAY[MIN_StationIndex..MAX_StationIndex] OF UDT_StationType;
  g_station_loc : ARRAY[1..MAX_StationIndex] OF UDT_UnitLocation;
  g_cfg         : ARRAY[1..MAX_Transporters] OF UDT_TransporterType;
  g_task        : ARRAY[1..MAX_Transporters] OF UDT_JC_TskQueueType;
  g_move        : ARRAY[1..MAX_Transporters] OF UDT_JC_MoveTimesType;
END_VAR
VAR
  ui       : INT;     (* unit loop *)
  qi       : INT;     (* queue index *)
  loc      : INT;     (* unit location station *)
  tgt      : INT;     (* unit target *)
  cov_t    : INT;     (* transporter loop *)
  ai       : INT;     (* task_area loop *)
  covers   : BOOL;    (* transporter covers this station *)
  done     : BOOL;    (* task created for this unit *)
  dest     : UDT_JC_NttDestType;  (* destination descriptor for this target+transporter *)
  ntt_idx  : INT;     (* resolved NTT index (maps TO_BUFFER to 6/7/8 based on batch) *)
  (* Location classification *)
  on_primary  : BOOL;  (* unit is already on a primary station *)
  on_fallback : BOOL;  (* unit is on a fallback station *)
  primary_free : BOOL; (* at least one primary station is free *)
  (* Destination search *)
  dest_stn : INT;     (* destination station *)
  si       : INT;     (* station loop *)
  station_idx      : INT;     (* candidate station *)
  stn_free : BOOL;
  uj       : INT;     (* inner unit loop for free check *)
  (* Duplicate check *)
  ti       : INT;     (* inner transporter loop *)
  already  : BOOL;    (* unit already queued or being transported *)
  qi2      : INT;     (* queue scan index *)
  (* Timing *)
  xfer_s   : REAL;    (* total transfer time *)
  task_start : LINT;
  task_end   : LINT;
  (* Idle-slot overlap check *)
  has_overlap    : BOOL;
  ntt_start      : LINT;
  ntt_end        : LINT;
  ov_s           : LINT;
  ov_e           : LINT;
  margin_travel  : REAL;
  slot_start     : LINT;   (* idle slot bounds *)
  tmp_move       : UDT_JC_MoveTimesType;  (* MATIEC cannot index arrays in FUNCTION args *)
  slot_end       : LINT;
  earliest_start : LINT;   (* earliest NTT start considering travel *)
  latest_end     : LINT;   (* latest NTT end considering travel *)
  travel_to_lift : REAL;
  travel_from_sink : REAL;
  ntt_duration   : LINT;
  qi3            : INT;   (* queue loop for idle-slot calc *)
  slot_ok        : BOOL;
  sh             : INT;   (* shift loop for insert-at-first *)
  (* Multi-transporter shared-area idle check *)
  ot             : INT;   (* other transporter loop *)
  oq             : INT;   (* other transporter queue loop *)
  overlap_conflict : BOOL;
  dest_x         : DINT;  (* dest_stn X position mm *)
  avoid_dist     : DINT;  (* cov_t avoid distance mm *)
  cov_min_x      : DINT;  (* cov_t drive limit min mm *)
  cov_max_x      : DINT;  (* cov_t drive limit max mm *)
  ot_min_x       : DINT;  (* other transporter drive limit min mm *)
  ot_max_x       : DINT;  (* other transporter drive limit max mm *)
  zone_min_x     : DINT;  (* shared overlap zone min mm *)
  zone_max_x     : DINT;  (* shared overlap zone max mm *)
  danger_min     : DINT;  (* zone_min - avoid_dist *)
  danger_max     : DINT;  (* zone_max + avoid_dist *)
  (* Shared-area timing: NTT split into own-area + shared-area portions *)
  loc_idx        : INT;   (* from_stn index = loc - 100 *)
  loc_x          : DINT;  (* lift station X position mm *)
  phase2_s       : REAL;  (* Phase 2 duration: lift + drip + tray (own area time) *)
  shared_entry   : LINT;  (* time when NTT enters shared area *)
  shared_time    : REAL;  (* duration NTT is on shared area *)
  ot_idle_ok     : BOOL;  (* other transporter has sufficient idle window *)
  ot_idle_start  : LINT;  (* other transporter idle window start *)
  ot_idle_end    : LINT;  (* other transporter idle window end *)
END_VAR

FOR ui := 1 TO MAX_Units DO
  tgt := g_unit[ui].Target;
  loc := g_unit[ui].location;

  (* Skip: no target, not on station.
     TO_PROCESS(3) is only handled here when batch state = NOT_PROCESSED
     (loaded unit waiting for processing → route to loaded-buffer). *)
  IF tgt >= 1 AND tgt <= 5 AND loc >= 100 THEN

    (* TO_PROCESS with batch already IN_PROCESS or later → skip (handled by schedule) *)
    IF tgt = 3 AND (g_batch[ui].BatchCode = 0 OR g_batch[ui].State <> 0) THEN
      CONTINUE;
    END_IF;

    (* Skip if unit already has a pending task in any queue or is being transported *)
    already := FALSE;
    FOR ti := 1 TO MAX_Transporters DO
      IF NOT already THEN
        (* Being transported right now? *)
        IF g_transporter[ti].Phase > 0 AND g_station_loc[ti].UnitId = ui THEN
          already := TRUE;
        END_IF;
        (* In any task queue? *)
        FOR qi2 := 1 TO g_task[ti].Count DO
          IF NOT already THEN
            IF g_task[ti].Queue[qi2].Unit = ui THEN
              already := TRUE;
            END_IF;
          END_IF;
        END_FOR;
      END_IF;
    END_FOR;

    IF NOT already THEN

    (* Try each transporter — not just the first covering one *)
    done := FALSE;
    FOR cov_t := 1 TO MAX_Transporters DO
      IF NOT done THEN

      (* Check coverage: transporter task_area covers this station *)
      covers := FALSE;
      FOR ai := 1 TO 4 DO
        IF NOT covers THEN
          IF g_cfg[cov_t].TaskArea[ai].MinLift > 0 OR g_cfg[cov_t].TaskArea[ai].MaxLift > 0 THEN
            IF loc >= g_cfg[cov_t].TaskArea[ai].MinLift AND loc <= g_cfg[cov_t].TaskArea[ai].MaxLift THEN
              covers := TRUE;
            END_IF;
          END_IF;
        END_IF;
      END_FOR;

      IF covers AND g_transporter[cov_t].IsActive
         AND (g_transporter[cov_t].Phase = 0 OR tgt = 5) THEN

        (* ── Resolve NTT index ── *)
        (* TO_BUFFER(2) maps to 6/7/8 depending on batch state *)
        (* TO_PROCESS(3) with NOT_PROCESSED batch → loaded buffer (7) *)
        IF tgt = 2 THEN
          IF g_batch[ui].BatchCode = 0 THEN
            ntt_idx := 6;  (* empty buffer — no batch *)
          ELSIF g_batch[ui].State = 2 THEN
            ntt_idx := 8;  (* processed buffer — batch PROCESSED *)
          ELSE
            ntt_idx := 7;  (* loaded buffer — batch NOT_PROCESSED or IN_PROCESS *)
          END_IF;
        ELSIF tgt = 3 THEN
          ntt_idx := 7;    (* TO_PROCESS + NOT_PROCESSED → loaded buffer *)
        ELSE
          ntt_idx := tgt;  (* other targets use their code directly *)
        END_IF;

        (* Get destination descriptor for this target + transporter *)
        dest := g_ntt[cov_t].Target[ntt_idx];

        (* ── Classify current location ── *)
        on_primary := FALSE;
        FOR si := 1 TO dest.StationCount DO
          IF dest.Stations[si] = loc THEN
            on_primary := TRUE;
          END_IF;
        END_FOR;

        (* Already on a primary station → no move needed *)
        IF NOT on_primary THEN

          on_fallback := FALSE;
          FOR si := 1 TO dest.FallbackCount DO
            IF dest.FallbackStations[si] = loc THEN
              on_fallback := TRUE;
            END_IF;
          END_FOR;

          (* Check if any primary station is free *)
          primary_free := FALSE;
          FOR si := 1 TO dest.StationCount DO
            station_idx := dest.Stations[si];
            IF station_idx <> loc AND station_idx >= MIN_StationIndex AND station_idx <= MAX_StationIndex THEN
              stn_free := TRUE;
              FOR uj := 1 TO MAX_Units DO
                IF g_unit[uj].location = station_idx AND g_unit[uj].Status = 1 THEN
                  stn_free := FALSE;
                END_IF;
              END_FOR;
              IF stn_free THEN
                primary_free := TRUE;
              END_IF;
            END_IF;
          END_FOR;

          dest_stn := 0;

          IF on_fallback AND NOT primary_free THEN
            (* On fallback, no primary free → stay put, don't bounce *)
            dest_stn := 0;
          ELSIF on_fallback AND primary_free THEN
            (* On fallback, primary is free → move to primary *)
            FOR si := 1 TO dest.StationCount DO
              IF dest_stn = 0 THEN
                station_idx := dest.Stations[si];
                IF station_idx <> loc AND station_idx >= MIN_StationIndex AND station_idx <= MAX_StationIndex THEN
                  stn_free := TRUE;
                  FOR uj := 1 TO MAX_Units DO
                    IF g_unit[uj].location = station_idx AND g_unit[uj].Status = 1 THEN
                      stn_free := FALSE;
                    END_IF;
                  END_FOR;
                  IF stn_free THEN
                    dest_stn := station_idx;
                  END_IF;
                END_IF;
              END_IF;
            END_FOR;
          ELSE
            (* Not on any known destination → full search: primary then fallback *)
            FOR si := 1 TO dest.StationCount DO
              IF dest_stn = 0 THEN
                station_idx := dest.Stations[si];
                IF station_idx <> loc AND station_idx >= MIN_StationIndex AND station_idx <= MAX_StationIndex THEN
                  stn_free := TRUE;
                  FOR uj := 1 TO MAX_Units DO
                    IF g_unit[uj].location = station_idx AND g_unit[uj].Status = 1 THEN
                      stn_free := FALSE;
                    END_IF;
                  END_FOR;
                  IF stn_free THEN
                    dest_stn := station_idx;
                  END_IF;
                END_IF;
              END_IF;
            END_FOR;

            IF dest_stn = 0 THEN
              FOR si := 1 TO dest.FallbackCount DO
                IF dest_stn = 0 THEN
                  station_idx := dest.FallbackStations[si];
                  IF station_idx <> loc AND station_idx >= MIN_StationIndex AND station_idx <= MAX_StationIndex THEN
                    stn_free := TRUE;
                    FOR uj := 1 TO MAX_Units DO
                      IF g_unit[uj].location = station_idx AND g_unit[uj].Status = 1 THEN
                        stn_free := FALSE;
                      END_IF;
                    END_FOR;
                    IF stn_free THEN
                      dest_stn := station_idx;
                    END_IF;
                  END_IF;
                END_IF;
              END_FOR;
            END_IF;
          END_IF;

          IF dest_stn > 0 THEN
            (* Calculate timing *)
            tmp_move := g_move[cov_t];
            xfer_s := STC_CalcTransferTime(
              i_from_stn            := loc,
              i_to_stn              := dest_stn,
              i_move                := tmp_move,
              i_from_dropping_x10   := g_station[loc].DrippingTime,
              i_to_device_delay_x10 := g_station[dest_stn].DeviceDelay,
              i_drip_tray_delay_x10 := g_cfg[cov_t].DripTrayDelay
            );

            task_start := i_time_s;
            task_end   := task_start + REAL_TO_LINT(xfer_s);
            ntt_duration := task_end - task_start;

            (* ── Current-slot check: NTT fits only in the CURRENT idle slot ──
               Like JS: find the slot where start <= now < end, check totalTime
               fits. NTT is never placed into future slots — only "right now". *)
            slot_ok := FALSE;

            IF g_task[cov_t].Count = 0 THEN
              (* No existing tasks → NTT always fits *)
              slot_ok := TRUE;
            ELSE
              (* Current slot = time from NOW until first queued task starts.
                 NTT must fit: task_end + travel_to_next_lift <= queue[1].StartTime *)
              IF g_task[cov_t].Queue[1].StartTime > task_start THEN
                slot_start := task_start;
                slot_end   := g_task[cov_t].Queue[1].StartTime;
                (* Travel from NTT sink to first task's lift *)
                travel_from_sink := STC_CalcHorizontalTravel(
                  i_from_stn := dest_stn,
                  i_to_stn   := g_task[cov_t].Queue[1].LiftStationTarget,
                  i_move     := g_move[cov_t]
                );
                latest_end := slot_end - REAL_TO_LINT(travel_from_sink) - 1;
                IF task_start >= slot_start AND task_end <= latest_end THEN
                  slot_ok := TRUE;
                END_IF;
              END_IF;
            END_IF;

            IF NOT slot_ok THEN
              (* Exception: if the next queued task's sink station is where
                 this NTT unit sits, we MUST move it first or we deadlock.
                 Force-insert; future scheduling will re-stabilize the list. *)
              IF g_task[cov_t].Count > 0
                 AND g_task[cov_t].Queue[1].SinkStationTarget = loc THEN
                slot_ok := TRUE;  (* force — deadlock prevention *)
              ELSE
                dest_stn := 0;  (* NTT doesn't fit → skip *)
              END_IF;
            END_IF;
          END_IF;

          (* ── Multi-transporter shared-area idle check ──
             If dest_stn is on the shared drive area between two transporters,
             the other transporter must have an idle window covering the time
             when THIS transporter is physically on the shared area.

             NTT transfer phases:
               Phase 2: lift + drip + tray  (nostin on vielä lift-asemalla)
               Phase 3: horizontal travel   (nostin liikkuu kohti dest)
               Phase 4: lower + tray + dev  (nostin on dest-asemalla)

             If lift station is NOT on shared area:
               shared_entry = task_start + phase2_s  (travel starts)
               shared_time  = xfer_s - phase2_s
             If lift station IS on shared area:
               shared_entry = task_start  (already there)
               shared_time  = xfer_s
          *)
          IF dest_stn > 0 THEN
            overlap_conflict := FALSE;
            dest_x := g_station[dest_stn].XPosition;
            avoid_dist := g_cfg[cov_t].AvoidanceWidth;
            cov_min_x := g_cfg[cov_t].DrivePosMin;
            cov_max_x := g_cfg[cov_t].DrivePosMax;

            FOR ot := 1 TO MAX_Transporters DO
              IF ot <> cov_t AND NOT overlap_conflict
                 AND g_transporter[ot].IsActive THEN
                ot_min_x := g_cfg[ot].DrivePosMin;
                ot_max_x := g_cfg[ot].DrivePosMax;

                (* Shared drive overlap zone *)
                IF cov_min_x > ot_min_x THEN zone_min_x := cov_min_x;
                ELSE zone_min_x := ot_min_x; END_IF;
                IF cov_max_x < ot_max_x THEN zone_max_x := cov_max_x;
                ELSE zone_max_x := ot_max_x; END_IF;

                IF zone_min_x >= zone_max_x THEN
                  CONTINUE; (* No drive overlap → no conflict possible *)
                END_IF;

                (* Is dest_stn in the overlap zone? *)
                IF dest_x < zone_min_x OR dest_x > zone_max_x THEN
                  CONTINUE; (* dest outside shared area *)
                END_IF;

                (* Danger zone = overlap ± avoid_distance *)
                danger_min := zone_min_x - avoid_dist;
                danger_max := zone_max_x + avoid_dist;

                (* ── Calculate shared-area entry time and duration ── *)
                loc_x := g_station[loc].XPosition;
                IF loc_x >= danger_min AND loc_x <= danger_max THEN
                  (* Lift station is ALSO on shared area → entire NTT *)
                  shared_entry := task_start;
                  shared_time  := xfer_s;
                ELSE
                  (* Lift station is on own area → shared starts after Phase 2 *)
                  loc_idx := loc - 100;
                  IF loc_idx >= 1 AND loc_idx <= 25 THEN
                    phase2_s := INT_TO_REAL(g_move[cov_t].LiftTime[loc_idx]) / 10.0
                              + INT_TO_REAL(g_station[loc].DrippingTime) / 10.0
                              + INT_TO_REAL(g_cfg[cov_t].DripTrayDelay) / 10.0;
                  ELSE
                    phase2_s := 0.0;
                  END_IF;
                  shared_entry := task_start + REAL_TO_LINT(phase2_s);
                  shared_time  := xfer_s - phase2_s;
                  IF shared_time < 1.0 THEN shared_time := 1.0; END_IF;
                END_IF;

                (* ── Check: does other transporter have an idle window
                     that starts ≤ shared_entry and lasts ≥ shared_time? ── *)
                ot_idle_ok := FALSE;

                IF g_task[ot].Count = 0 AND g_transporter[ot].Phase = 0 THEN
                  (* Other transporter fully idle → OK *)
                  ot_idle_ok := TRUE;
                ELSE
                  (* Find idle window covering shared_entry..shared_entry+shared_time *)

                  (* Window before first queued task *)
                  IF g_task[ot].Count > 0 THEN
                    (* Idle starts: now (or after active task finishes) *)
                    IF g_transporter[ot].Phase >= 1 AND g_transporter[ot].Phase <= 4 THEN
                      ot_idle_start := g_task[ot].Queue[1].FinishTime;
                    ELSE
                      ot_idle_start := task_start;  (* idle now *)
                    END_IF;
                    ot_idle_end := g_task[ot].Queue[1].StartTime;
                    IF ot_idle_start <= shared_entry
                       AND ot_idle_end >= shared_entry + REAL_TO_LINT(shared_time) THEN
                      ot_idle_ok := TRUE;
                    END_IF;
                  END_IF;

                  (* Windows between consecutive queued tasks *)
                  IF NOT ot_idle_ok THEN
                    FOR oq := 1 TO g_task[ot].Count - 1 DO
                      IF NOT ot_idle_ok THEN
                        ot_idle_start := g_task[ot].Queue[oq].FinishTime;
                        ot_idle_end   := g_task[ot].Queue[oq + 1].StartTime;
                        IF ot_idle_start <= shared_entry
                           AND ot_idle_end >= shared_entry + REAL_TO_LINT(shared_time) THEN
                          ot_idle_ok := TRUE;
                        END_IF;
                      END_IF;
                    END_FOR;
                  END_IF;

                  (* Window after last queued task *)
                  IF NOT ot_idle_ok AND g_task[ot].Count > 0 THEN
                    ot_idle_start := g_task[ot].Queue[g_task[ot].Count].FinishTime;
                    IF ot_idle_start <= shared_entry THEN
                      ot_idle_ok := TRUE;  (* open-ended idle after last task *)
                    END_IF;
                  END_IF;
                END_IF;

                IF NOT ot_idle_ok THEN
                  overlap_conflict := TRUE;
                END_IF;
              END_IF;
            END_FOR;

            IF overlap_conflict THEN
              dest_stn := 0;
            END_IF;
          END_IF;

          IF dest_stn > 0 THEN
            (* Insert as FIRST task — shift existing tasks down *)
            IF g_task[cov_t].Count < MAX_TASK_QUEUE THEN
              (* Shift queue[1..Count] → queue[2..Count+1] *)
              FOR sh := g_task[cov_t].Count TO 1 BY -1 DO
                g_task[cov_t].Queue[sh + 1] := g_task[cov_t].Queue[sh];
              END_FOR;
              g_task[cov_t].Queue[1].Unit         := ui;
              g_task[cov_t].Queue[1].Stage        := 0;  (* no program stage *)
              g_task[cov_t].Queue[1].LiftStationTarget := loc;
              g_task[cov_t].Queue[1].SinkStationTarget := dest_stn;
              g_task[cov_t].Queue[1].StartTime   := task_start;
              g_task[cov_t].Queue[1].FinishTime  := task_end;
              g_task[cov_t].Queue[1].CalcTime    := 0;
              g_task[cov_t].Queue[1].MinTime     := 0;
              g_task[cov_t].Queue[1].MaxTime     := 0;
              (* Check if dest_stn is a primary station for this NTT target *)
              g_task[cov_t].Queue[1].NttPrimary := 0;
              FOR si := 1 TO dest.StationCount DO
                IF dest.Stations[si] = dest_stn THEN
                  g_task[cov_t].Queue[1].NttPrimary := 1;
                END_IF;
              END_FOR;
              g_task[cov_t].Count := g_task[cov_t].Count + 1;
              done := TRUE;
            END_IF;
          END_IF;

        END_IF; (* NOT on_primary *)

      END_IF; (* covers + idle *)

      END_IF; (* NOT done *)
    END_FOR; (* transporter loop *)

    END_IF; (* NOT already *)

  END_IF; (* valid target *)
END_FOR;

END_FUNCTION_BLOCK

(* ---- TSK_FB_Resolve.st ---- *)
(* ============================================================
   TSK_FB_Resolve — Conflict resolution matching JS resolveConflict()
   ============================================================
   Ported from transporterTaskScheduler.js resolveConflict() (line 1638)

   Four sequential phases — each reduces remaining deficit,
   next phase uses the remainder (partial solutions accumulate):

     Phase 1: ADVANCE — advance blocked batch using
              CHAIN bottleneck + SUFFIX flex_down
              (walks backward through earlier stages)
     Phase 2: DELAY   — delay conflict batch using
              SINGLE-STAGE flex_up (conf_stage only)
     Phase 3: PRECEDING_DELAY — delay conf batch at stage-1
     Phase 4: DELAY_PREV_PAST_NEXT — delay blocked batch to
              force order swap (only if NOT swappable)

   lockedStages prevents oscillation: once a stage is advanced,
   it cannot be delayed, and vice versa.

   Cap factor: 90% if batch is on that stage, 50% otherwise.

   Each phase applies a FLAT SHIFT: modify the target stage's
   CalcTime + ExitTime, then fb_shift propagates to subsequent
   stages and task queue entries.

   The caller loop (TSK_FB_Scheduler 2200→2202→2203) re-runs
   SORT → SWAP → ANALYZE after each resolve, so partial
   solutions converge over iterations.
   ============================================================ *)

FUNCTION_BLOCK TSK_FB_Resolve
VAR_INPUT
  i_conf_unit     : INT;     (* conflict task: unit *)
  i_conf_stage    : INT;     (* conflict task: stage *)
  i_conf_trans    : INT;     (* conflict task: transporter *)
  i_blocked_unit  : INT;     (* blocking task: unit *)
  i_blocked_stage : INT;     (* blocking task: stage *)
  i_deficit       : REAL;    (* seconds short *)
END_VAR
VAR_IN_OUT
  io_locks    : ARRAY[1..50] OF UDT_JC_TskLockType;
  io_lock_cnt : INT;
END_VAR
VAR_EXTERNAL CONSTANT
    MAX_Transporters : INT;
    MAX_Units        : INT;
END_VAR

VAR_EXTERNAL
  g_task    : ARRAY[1..MAX_Transporters] OF UDT_JC_TskQueueType;
  g_schedule : ARRAY[1..MAX_Units] OF UDT_JC_TskScheduleType;
  g_batch   : ARRAY[1..MAX_Units] OF UDT_BatchType;
END_VAR
VAR_OUTPUT
  o_solved      : BOOL;
  o_total_delay : REAL;
  o_total_adv   : REAL;
END_VAR
VAR
  remain      : REAL;
  cap         : REAL;
  amount      : REAL;
  stage_flex  : REAL;
  (* Lock checking *)
  is_locked_adv   : BOOL;   (* blocked stage locked DELAY → cannot ADVANCE *)
  is_locked_del   : BOOL;   (* conf stage locked ADVANCE → cannot DELAY *)
  can_advance     : BOOL;
  can_delay       : BOOL;
  lock_i          : INT;
  (* Priority 3 — PRECEDING_DELAY *)
  prev_conf_stage   : INT;
  is_pcs_locked     : BOOL;
  (* Priority 4 — DELAY_PREV_PAST_NEXT *)
  prev_sink_stn     : INT;
  next_lift_stn     : INT;
  is_blk_adv_locked : BOOL;
  qi                : INT;
  (* Chain advance — JS: walk backward to find bottleneck *)
  chain_flex     : REAL;   (* bottleneck flex among earlier stages *)
  suffix_flex    : REAL;   (* conflictFlexDown - chainFlexDown *)
  earlier_stg    : INT;    (* loop variable for chain walk *)
  earlier_flex   : REAL;   (* individual earlier stage flex_down *)
  chain_amount   : REAL;   (* amount from CHAIN_ADVANCE *)
  suffix_amount  : REAL;   (* amount from SUFFIX_ADVANCE *)
  (* Shared shift FB *)
  fb_shift : STC_FB_ShiftSchedule;
END_VAR

o_solved      := FALSE;
o_total_delay := 0.0;
o_total_adv   := 0.0;
remain        := i_deficit;

IF remain <= 0.1 THEN
  o_solved := TRUE;
  RETURN;
END_IF;

(* ══════ Lock check: is blocked stage locked DELAY? (cannot ADVANCE) ══════ *)
is_locked_adv := FALSE;
FOR lock_i := 1 TO io_lock_cnt DO
  IF io_locks[lock_i].Unit = i_blocked_unit
     AND io_locks[lock_i].Stage = i_blocked_stage
     AND io_locks[lock_i].Direction = 2 THEN  (* 2=DELAY *)
    is_locked_adv := TRUE;
  END_IF;
END_FOR;

(* ══════ Lock check: is conf stage locked ADVANCE? (cannot DELAY) ══════ *)
is_locked_del := FALSE;
FOR lock_i := 1 TO io_lock_cnt DO
  IF io_locks[lock_i].Unit = i_conf_unit
     AND io_locks[lock_i].Stage = i_conf_stage
     AND io_locks[lock_i].Direction = 1 THEN  (* 1=ADVANCE *)
    is_locked_del := TRUE;
  END_IF;
END_FOR;

can_advance := NOT is_locked_adv;
can_delay   := NOT is_locked_del;

(* ══════════════════════════════════════════════════════════════ *)
(* PHASE 1: ADVANCE — advance blocked batch (JS Vaihe 1)       *)
(* Chain bottleneck: walk backward through earlier stages to    *)
(* find smallest flex_down < conflictFlexDown.                  *)
(* CHAIN_ADVANCE uses bottleneck, SUFFIX_ADVANCE uses remainder *)
(* JS: resolveConflict() lines 1738-1860                        *)
(* ══════════════════════════════════════════════════════════════ *)
IF can_advance
   AND i_blocked_unit >= 1 AND i_blocked_unit <= MAX_Units
   AND i_blocked_stage >= 1 THEN
IF i_blocked_stage <= g_schedule[i_blocked_unit].StageCount THEN

  (* Conflict stage's own flex_down *)
  stage_flex := DINT_TO_REAL(
    g_schedule[i_blocked_unit].Stages[i_blocked_stage].CalcTime
    - g_schedule[i_blocked_unit].Stages[i_blocked_stage].MinTime);
  IF stage_flex < 0.0 THEN stage_flex := 0.0; END_IF;

  IF stage_flex > 0.1 THEN
    (* Cap: 90% if batch is on this stage, 50% otherwise *)
    IF g_batch[i_blocked_unit].CurStage = g_schedule[i_blocked_unit].Stages[i_blocked_stage].ProgramStage THEN
      cap := 0.9;
    ELSE
      cap := 0.5;
    END_IF;

    (* -- Chain bottleneck search -- *)
    (* JS: walk backward through prevBatchTasks (stages < conflictStage) *)
    (* Find smallest flex_down among earlier stages that is < conflictFlexDown *)
    chain_flex := stage_flex;  (* init to conflict stage flex = no bottleneck *)
    FOR earlier_stg := 1 TO i_blocked_stage - 1 DO
      earlier_flex := DINT_TO_REAL(
        g_schedule[i_blocked_unit].Stages[earlier_stg].CalcTime
        - g_schedule[i_blocked_unit].Stages[earlier_stg].MinTime);
      IF earlier_flex < 0.0 THEN earlier_flex := 0.0; END_IF;
      IF earlier_flex > 0.0 AND earlier_flex < chain_flex THEN
        chain_flex := earlier_flex;
      END_IF;
    END_FOR;
    (* If no earlier stage had positive flex < conflictFlex, chain_flex = stage_flex *)
    (* In that case suffix_flex = 0 and all advance comes from chain *)

    (* -- CHAIN_ADVANCE: apply bottleneck amount -- *)
    chain_amount := chain_flex * cap;
    IF chain_amount > remain THEN chain_amount := remain; END_IF;

    IF chain_amount > 0.1 THEN
      g_schedule[i_blocked_unit].Stages[i_blocked_stage].CalcTime :=
        g_schedule[i_blocked_unit].Stages[i_blocked_stage].CalcTime - REAL_TO_DINT(chain_amount);
      g_schedule[i_blocked_unit].Stages[i_blocked_stage].ExitTime :=
        g_schedule[i_blocked_unit].Stages[i_blocked_stage].ExitTime - REAL_TO_LINT(chain_amount);

      fb_shift(i_unit := i_blocked_unit, i_from_stage := i_blocked_stage + 1, i_amount := -chain_amount);

      g_batch[i_blocked_unit].CalTime :=
        g_batch[i_blocked_unit].CalTime - REAL_TO_DINT(chain_amount);
      IF g_batch[i_blocked_unit].CalTime < g_batch[i_blocked_unit].MinTime THEN
        g_batch[i_blocked_unit].CalTime := g_batch[i_blocked_unit].MinTime;
      END_IF;

      remain := remain - chain_amount;
      o_total_adv := o_total_adv + chain_amount;
    END_IF;

    (* -- SUFFIX_ADVANCE: use remaining flex beyond bottleneck -- *)
    (* JS: suffixFlexDown = conflictFlexDown - chainFlexDown *)
    suffix_flex := stage_flex - chain_flex;
    IF suffix_flex > 0.1 AND remain > 0.1 THEN
      suffix_amount := suffix_flex * cap;
      IF suffix_amount > remain THEN suffix_amount := remain; END_IF;

      IF suffix_amount > 0.1 THEN
        g_schedule[i_blocked_unit].Stages[i_blocked_stage].CalcTime :=
          g_schedule[i_blocked_unit].Stages[i_blocked_stage].CalcTime - REAL_TO_DINT(suffix_amount);
        g_schedule[i_blocked_unit].Stages[i_blocked_stage].ExitTime :=
          g_schedule[i_blocked_unit].Stages[i_blocked_stage].ExitTime - REAL_TO_LINT(suffix_amount);

        fb_shift(i_unit := i_blocked_unit, i_from_stage := i_blocked_stage + 1, i_amount := -suffix_amount);

        g_batch[i_blocked_unit].CalTime :=
          g_batch[i_blocked_unit].CalTime - REAL_TO_DINT(suffix_amount);
        IF g_batch[i_blocked_unit].CalTime < g_batch[i_blocked_unit].MinTime THEN
          g_batch[i_blocked_unit].CalTime := g_batch[i_blocked_unit].MinTime;
        END_IF;

        remain := remain - suffix_amount;
        o_total_adv := o_total_adv + suffix_amount;
      END_IF;
    END_IF;

    (* Record lock: ADVANCE on blocked stage *)
    IF io_lock_cnt < 50 THEN
      io_lock_cnt := io_lock_cnt + 1;
      io_locks[io_lock_cnt].Unit := i_blocked_unit;
      io_locks[io_lock_cnt].Stage := i_blocked_stage;
      io_locks[io_lock_cnt].Direction := 1;  (* 1=ADVANCE *)
    END_IF;

    IF remain <= 0.1 THEN
      o_solved := TRUE;
      RETURN;
    END_IF;
  END_IF;
END_IF;
END_IF;

(* ══════════════════════════════════════════════════════════════ *)
(* PHASE 2: DELAY — delay conflict batch (JS Vaihe 2)          *)
(* Single-stage flex: conf_stage MaxTime - CalcTime             *)
(* Flat shift applied to conf_stage onward.                     *)
(* Partial delay is OK — remainder goes to Phase 3.             *)
(* ══════════════════════════════════════════════════════════════ *)
IF can_delay AND remain > 0.1
   AND i_conf_unit >= 1 AND i_conf_unit <= MAX_Units
   AND i_conf_stage >= 1 THEN
IF i_conf_stage <= g_schedule[i_conf_unit].StageCount THEN

  stage_flex := DINT_TO_REAL(
    g_schedule[i_conf_unit].Stages[i_conf_stage].MaxTime
    - g_schedule[i_conf_unit].Stages[i_conf_stage].CalcTime);
  IF stage_flex < 0.0 THEN stage_flex := 0.0; END_IF;

  IF stage_flex > 0.1 THEN
    IF g_batch[i_conf_unit].CurStage = g_schedule[i_conf_unit].Stages[i_conf_stage].ProgramStage THEN
      cap := 0.9;
    ELSE
      cap := 0.5;
    END_IF;
    amount := stage_flex * cap;
    IF amount > remain THEN amount := remain; END_IF;

    (* Apply: increase CalcTime of conf_stage *)
    g_schedule[i_conf_unit].Stages[i_conf_stage].CalcTime :=
      g_schedule[i_conf_unit].Stages[i_conf_stage].CalcTime + REAL_TO_DINT(amount);
    g_schedule[i_conf_unit].Stages[i_conf_stage].ExitTime :=
      g_schedule[i_conf_unit].Stages[i_conf_stage].ExitTime + REAL_TO_LINT(amount);

    fb_shift(i_unit := i_conf_unit, i_from_stage := i_conf_stage + 1, i_amount := amount);

    (* JS: propagateDelayToBatch updates batch.calc_time_s ONLY if batch is on this stage *)
    IF g_batch[i_conf_unit].CurStage = g_schedule[i_conf_unit].Stages[i_conf_stage].ProgramStage THEN
      g_batch[i_conf_unit].CalTime :=
        g_batch[i_conf_unit].CalTime + REAL_TO_DINT(amount);
      IF g_batch[i_conf_unit].CalTime > g_batch[i_conf_unit].MaxTime THEN
        g_batch[i_conf_unit].CalTime := g_batch[i_conf_unit].MaxTime;
      END_IF;
    END_IF;

    remain := remain - amount;
    o_total_delay := o_total_delay + amount;

    (* Record lock: DELAY on conf stage *)
    IF io_lock_cnt < 50 THEN
      io_lock_cnt := io_lock_cnt + 1;
      io_locks[io_lock_cnt].Unit := i_conf_unit;
      io_locks[io_lock_cnt].Stage := i_conf_stage;
      io_locks[io_lock_cnt].Direction := 2;  (* 2=DELAY *)
    END_IF;

    IF remain <= 0.1 THEN
      o_solved := TRUE;
      RETURN;
    END_IF;
  END_IF;
END_IF;
END_IF;

(* ══════════════════════════════════════════════════════════════ *)
(* PHASE 3: PRECEDING_DELAY — delay conf batch at stage-1       *)
(* (JS Vaihe 3)                                                 *)
(* Delay the conf batch's PREVIOUS stage to push everything     *)
(* ══════════════════════════════════════════════════════════════ *)
prev_conf_stage := i_conf_stage - 1;
IF remain > 0.1 AND prev_conf_stage >= 1 AND i_conf_unit >= 1 AND i_conf_unit <= MAX_Units THEN
  (* Check lock: is prev_conf_stage locked ADVANCE? → cannot DELAY *)
  is_pcs_locked := FALSE;
  FOR lock_i := 1 TO io_lock_cnt DO
    IF io_locks[lock_i].Unit = i_conf_unit
       AND io_locks[lock_i].Stage = prev_conf_stage
       AND io_locks[lock_i].Direction = 1 THEN
      is_pcs_locked := TRUE;
    END_IF;
  END_FOR;

  IF NOT is_pcs_locked THEN
    stage_flex := DINT_TO_REAL(g_schedule[i_conf_unit].Stages[prev_conf_stage].MaxTime
                - g_schedule[i_conf_unit].Stages[prev_conf_stage].CalcTime);
    IF stage_flex < 0.0 THEN stage_flex := 0.0; END_IF;

    IF stage_flex > 0.1 THEN
      IF g_batch[i_conf_unit].CurStage = g_schedule[i_conf_unit].Stages[prev_conf_stage].ProgramStage THEN
        cap := 0.9;
      ELSE
        cap := 0.5;
      END_IF;
      amount := stage_flex * cap;
      IF amount > remain THEN amount := remain; END_IF;

      g_schedule[i_conf_unit].Stages[prev_conf_stage].CalcTime :=
        g_schedule[i_conf_unit].Stages[prev_conf_stage].CalcTime + REAL_TO_DINT(amount);
      g_schedule[i_conf_unit].Stages[prev_conf_stage].ExitTime :=
        g_schedule[i_conf_unit].Stages[prev_conf_stage].ExitTime + REAL_TO_LINT(amount);
      fb_shift(i_unit := i_conf_unit, i_from_stage := prev_conf_stage + 1, i_amount := amount);

      (* JS: propagateDelayToBatch with propagateFromStage=conf_stage
         updates batch.calc_time_s ONLY if batch is on conf_stage *)
      IF g_batch[i_conf_unit].CurStage = g_schedule[i_conf_unit].Stages[i_conf_stage].ProgramStage THEN
        g_batch[i_conf_unit].CalTime :=
          g_batch[i_conf_unit].CalTime + REAL_TO_DINT(amount);
        IF g_batch[i_conf_unit].CalTime > g_batch[i_conf_unit].MaxTime THEN
          g_batch[i_conf_unit].CalTime := g_batch[i_conf_unit].MaxTime;
        END_IF;
      END_IF;

      remain := remain - amount;
      o_total_delay := o_total_delay + amount;

      (* Record lock *)
      IF io_lock_cnt < 50 THEN
        io_lock_cnt := io_lock_cnt + 1;
        io_locks[io_lock_cnt].Unit := i_conf_unit;
        io_locks[io_lock_cnt].Stage := prev_conf_stage;
        io_locks[io_lock_cnt].Direction := 2;
      END_IF;

      IF remain <= 0.1 THEN
        o_solved := TRUE;
        RETURN;
      END_IF;
    END_IF;
  END_IF;
END_IF;

(* ══════════════════════════════════════════════════════════════ *)
(* PHASE 4: DELAY_PREV_PAST_NEXT — delay blocked batch to       *)
(* force order swap (JS Vaihe 4)                                *)
(* Only if NOT swappable: prev.sink ≠ next.lift                 *)
(* ══════════════════════════════════════════════════════════════ *)
IF remain > 0.1 AND i_blocked_unit >= 1 AND i_blocked_unit <= MAX_Units THEN
  (* Find blocked and conf tasks in queue to check swap condition *)
  prev_sink_stn := 0;
  next_lift_stn := 0;
  IF i_conf_trans >= 1 AND i_conf_trans <= MAX_Transporters THEN
    FOR qi := 1 TO g_task[i_conf_trans].Count DO
      IF g_task[i_conf_trans].Queue[qi].Unit = i_blocked_unit
         AND g_task[i_conf_trans].Queue[qi].Stage = i_blocked_stage THEN
        prev_sink_stn := g_task[i_conf_trans].Queue[qi].SinkStationTarget;
      END_IF;
      IF g_task[i_conf_trans].Queue[qi].Unit = i_conf_unit
         AND g_task[i_conf_trans].Queue[qi].Stage = i_conf_stage THEN
        next_lift_stn := g_task[i_conf_trans].Queue[qi].LiftStationTarget;
      END_IF;
    END_FOR;
  END_IF;

  (* Swap check: if prev.sink = next.lift → swappable, skip *)
  IF NOT (prev_sink_stn > 0 AND next_lift_stn > 0 AND prev_sink_stn = next_lift_stn) THEN
    (* Check lock: is blocked stage locked ADVANCE? → cannot DELAY *)
    is_blk_adv_locked := FALSE;
    FOR lock_i := 1 TO io_lock_cnt DO
      IF io_locks[lock_i].Unit = i_blocked_unit
         AND io_locks[lock_i].Stage = i_blocked_stage
         AND io_locks[lock_i].Direction = 1 THEN
        is_blk_adv_locked := TRUE;
      END_IF;
    END_FOR;

    IF NOT is_blk_adv_locked THEN
      stage_flex := DINT_TO_REAL(g_schedule[i_blocked_unit].Stages[i_blocked_stage].MaxTime
                  - g_schedule[i_blocked_unit].Stages[i_blocked_stage].CalcTime);
      IF stage_flex < 0.0 THEN stage_flex := 0.0; END_IF;

      IF stage_flex > 0.1 THEN
        IF g_batch[i_blocked_unit].CurStage = g_schedule[i_blocked_unit].Stages[i_blocked_stage].ProgramStage THEN
          cap := 0.9;
        ELSE
          cap := 0.5;
        END_IF;
        amount := stage_flex * cap;
        IF amount > remain THEN amount := remain; END_IF;

        g_schedule[i_blocked_unit].Stages[i_blocked_stage].CalcTime :=
          g_schedule[i_blocked_unit].Stages[i_blocked_stage].CalcTime + REAL_TO_DINT(amount);
        g_schedule[i_blocked_unit].Stages[i_blocked_stage].ExitTime :=
          g_schedule[i_blocked_unit].Stages[i_blocked_stage].ExitTime + REAL_TO_LINT(amount);
        fb_shift(i_unit := i_blocked_unit, i_from_stage := i_blocked_stage + 1, i_amount := amount);

        (* JS: propagateDelayToBatch updates batch.calc_time_s ONLY if batch is on this stage *)
        IF g_batch[i_blocked_unit].CurStage = g_schedule[i_blocked_unit].Stages[i_blocked_stage].ProgramStage THEN
          g_batch[i_blocked_unit].CalTime :=
            g_batch[i_blocked_unit].CalTime + REAL_TO_DINT(amount);
          IF g_batch[i_blocked_unit].CalTime > g_batch[i_blocked_unit].MaxTime THEN
            g_batch[i_blocked_unit].CalTime := g_batch[i_blocked_unit].MaxTime;
          END_IF;
        END_IF;

        remain := remain - amount;
        o_total_delay := o_total_delay + amount;

        (* Record lock: DELAY on blocked stage *)
        IF io_lock_cnt < 50 THEN
          io_lock_cnt := io_lock_cnt + 1;
          io_locks[io_lock_cnt].Unit := i_blocked_unit;
          io_locks[io_lock_cnt].Stage := i_blocked_stage;
          io_locks[io_lock_cnt].Direction := 2;
        END_IF;

        IF remain <= 0.1 THEN
          o_solved := TRUE;
          RETURN;
        END_IF;
      END_IF;
    END_IF;
  END_IF;
END_IF;

(* If not solved, partial resolution was applied *)

END_FUNCTION_BLOCK

(* ---- TSK_FB_Scheduler.st ---- *)
(* ===========================================================================================
 *  TSK_FB_Scheduler — Main task scheduler state machine
 *
 *  Company : Galvatek part of the John Cockerill Group
 *  Author  : Jarmo Piipponen
 *  Created : 25.03.2026
 *
 * -------------------------------------------------------------------------------------------
 *  One phase per PLC scan cycle.
 *
 *  Phase flow (structured by 100/1000 groups):
 *  0        STOPPED
 *  1        INIT             (collect active batches)
 *  2        NO_TREATMENT_STATES
 *  1000+i   CALC_SCHEDULE    (schedule for batch i, 0..batch_count-1)
 *  2000     CLEAR_TASKS      (clear task queues)
 *  2001+i   CREATE_TASKS     (tasks for batch i, 0..batch_count-1)
 *  2100     SORT_TASKS
 *  2101     SWAP_TASKS
 *  2102     ANALYZE          (→ 2103 if conflict, → 2200 if clean)
 *  2103     RESOLVE          (→ 2100 loop, or → 2200 if max iter)
 *  2200     NO_TREATMENT     (create no-treatment tasks)
 *  2201     APPLY_STRETCHES  (persist resolve decisions)
 *  10000    READY            (cycle complete)
 *  10001    CHECK_DEP_PENDING
 *  10002    RESTART          (→ 1)
 *
 *  Phase advancement:
 *  Default = phase + 1 (at end of function body).
 *  next_phase is set ONLY when jumping to a different group.
 *
 *  Conflict resolution: one conflict per cycle.
 *  If resolved → back to SORT (2100).
 *  If no conflict → NO_TREATMENT → READY.
 *  Max iterations to prevent infinite loops.
 *
 *  ------------------------------------------------------------------------------------------
 *
 *  Changes:
 *  25.03.2026 - Restructured: phase+1 default, idx from phase offset.
 *
 *
 *)

FUNCTION_BLOCK TSK_FB_Scheduler

(* Introduction of Variables ----------------------------------------------------------------*)

VAR_INPUT
  i_run                     : BOOL;    (* TRUE = run, FALSE = stop *)
  i_time_s                  : LINT;    (* current absolute time (s), unix seconds *)
END_VAR

VAR_EXTERNAL CONSTANT
    MAX_TRANSPORTERS        : INT;
    MAX_UNITS               : INT;
    MAX_LOCKS               : INT;
END_VAR

VAR_EXTERNAL
  g_batch                   : ARRAY[1..MAX_UNITS] OF UDT_BatchType;
  g_unit                    : ARRAY[1..MAX_UNITS] OF UDT_JC_UnitType;
  TreatmentPrograms                 : ARRAY[1..MAX_UNITS] OF UDT_TreatmentProgramType;
  g_task                    : ARRAY[1..MAX_TRANSPORTERS] OF UDT_JC_TskQueueType;
  g_schedule                : ARRAY[1..MAX_UNITS] OF UDT_JC_TskScheduleType;
  Transporters                     : ARRAY[0..MAX_TRANSPORTERS] OF UDT_TransporterType;
  (* DEP handshake *)
  g_dep_pending             : UDT_JC_DepPendingWriteType;
  g_conflict_resolved       : BOOL;
  g_tsk_stable              : BOOL;
  (* Debug observability *)
  g_dbg_tsk_conflict_type   : INT;
  g_dbg_tsk_conflict_iter   : INT;
  g_dbg_tsk_conf_unit       : INT;
  g_dbg_tsk_conf_stage      : INT;
  g_dbg_tsk_blocked_unit    : INT;
  g_dbg_tsk_blocked_stage   : INT;
  g_dbg_tsk_deficit         : DINT;
  g_dbg_tsk_stretch_cnt     : INT;
  g_dbg_tsk_total_adv       : DINT;
  g_dbg_tsk_total_delay     : DINT;
  g_dbg_prog_cal            : ARRAY[1..MAX_UNITS] OF DINT;
END_VAR

VAR_OUTPUT
  o_phase                   : INT;
  o_batch_cnt               : INT;
  o_task_cnt                : INT;
  o_cycle_cnt               : INT;
  o_conflict                : BOOL;
  o_round_ticks             : INT;     (* ticks consumed by last completed round *)
END_VAR

VAR
  phase                     : INT := 0;
  next_phase                : INT;
  idx                       : INT;    (* derived from phase offset *)
  (* Batch list *)
  batch_list                : ARRAY[1..MAX_UNITS] OF INT;
  batch_count               : INT;
  (* Conflict iteration *)
  conflict_iter             : INT;
  MAX_CONFLICT_ITER         : INT := 40;
  (* Analyze result cache *)
  an_conflict               : BOOL;
  an_conf_type              : INT;
  an_conf_unit              : INT;
  an_conf_stage             : INT;
  an_conf_trans             : INT;
  an_blocked_unit           : INT;
  an_blocked_stage          : INT;
  an_deficit                : REAL;
  (* Resolve result cache *)
  rs_total_adv              : REAL;
  rs_total_delay            : REAL;
  (* Transporter assignment *)
  sched_trans               : INT;
  (* Locked stages — prevents oscillation in resolve loop *)
  locks                     : ARRAY[1..MAX_LOCKS] OF UDT_JC_TskLockType;
  lock_cnt                  : INT := 0;
  locks_initialized         : BOOL := FALSE;
  fb_find                   : STC_FindTransporter;
  (* candidateStretches — JS: resolve decisions persisted to TreatmentPrograms *)
  stretches                 : ARRAY[1..20] OF UDT_JC_TskStretchType;
  stretch_cnt               : INT := 0;
  si                        : INT;
  new_cal                   : DINT;
  flex_cap                  : DINT;
  (* Temp *)
  ui                        : INT;
  ui2                       : INT;
  ti                        : INT;
  bi                        : INT;
  total_tasks               : INT;
  cycle_count               : INT := 0;
  round_ticks               : INT := 0;  (* ticks since last RESTART *)
END_VAR

IF NOT i_run THEN
  IF phase <> 0 THEN
    FOR ti := 1 TO MAX_TRANSPORTERS DO
      g_task[ti].Count := 0;
    END_FOR;
  END_IF;
  phase := 0;
  o_phase := 0;
  RETURN;
END_IF;

next_phase := 0;
round_ticks := round_ticks + 1;

(* ══════════════════════════════════════════════════════════════ *)
(* PHASE 0: STOPPED                                             *)
(* ══════════════════════════════════════════════════════════════ *)
IF phase = 0 THEN
  next_phase := 1;

(* ══════════════════════════════════════════════════════════════ *)
(* PHASE 1: INIT — collect active batches                       *)
(* ══════════════════════════════════════════════════════════════ *)
ELSIF phase = 1 THEN
  (* Clear schedule for ALL units — start from clean slate *)
  FOR ui := 1 TO MAX_UNITS DO
    g_schedule[ui].StageCount := 0;
  END_FOR;
  batch_count := STC_CollectActiveBatches(i_mode := 0, o_list => batch_list);
  o_batch_cnt := batch_count;
  conflict_iter := 0;
  locks_initialized := FALSE;
  stretch_cnt := 0;
  g_dbg_tsk_total_adv   := 0;
  g_dbg_tsk_total_delay := 0;

  IF batch_count = 0 THEN
    FOR ti := 1 TO MAX_TRANSPORTERS DO
      g_task[ti].Count := 0;
    END_FOR;
    g_conflict_resolved := TRUE;
    next_phase := 2200;   (* skip to NO_TREATMENT *)
  ELSE
    g_conflict_resolved := FALSE;
    (* phase + 1 → 2 *)
  END_IF;

(* ══════════════════════════════════════════════════════════════ *)
(* PHASE 2: NO_TREATMENT_STATES                                *)
(* ══════════════════════════════════════════════════════════════ *)
ELSIF phase = 2 THEN
  STC_NoTreatmentStates();
  next_phase := 1000;

(* ══════════════════════════════════════════════════════════════ *)
(* PHASE 1000+i: CALC_SCHEDULE — one batch per scan             *)
(*   i = 0..batch_count-1: calculate schedule                   *)
(*   i >= batch_count: done → 2000                              *)
(* ══════════════════════════════════════════════════════════════ *)
ELSIF phase >= 1000 AND phase <= 1999 THEN
  idx := phase - 1000;

  IF idx < batch_count THEN
    ui := batch_list[idx + 1];

    (* CalcSchedule handles elapsed-time normalisation — no pre-adjustment needed here. *)

    IF g_unit[ui].location < MIN_STATION_INDEX THEN
      sched_trans := g_unit[ui].location;
    ELSE
      fb_find(i_lift_stn := g_unit[ui].location, i_sink_stn := 0);
      sched_trans := fb_find.o_trans;
      IF sched_trans = 0 THEN sched_trans := 1; END_IF;
    END_IF;

    STC_CalcSchedule(i_unit := ui, i_trans := sched_trans, i_time_s := i_time_s,
                     io_schedule := g_schedule, io_batch := g_batch, io_program := TreatmentPrograms);
    (* phase + 1 → next batch *)

  ELSE
    next_phase := 2000;
  END_IF;

(* ══════════════════════════════════════════════════════════════ *)
(* PHASE 2000: CLEAR_TASKS — clear all task queues              *)
(* ══════════════════════════════════════════════════════════════ *)
ELSIF phase = 2000 THEN
  FOR ti := 1 TO MAX_TRANSPORTERS DO
    g_task[ti].Count := 0;
  END_FOR;
  (* phase + 1 → 2001 *)

(* ══════════════════════════════════════════════════════════════ *)
(* PHASE 2001+i: CREATE_TASKS — one batch per scan              *)
(*   i = 0..batch_count-1: create tasks                         *)
(*   i >= batch_count: done → 2100                              *)
(* ══════════════════════════════════════════════════════════════ *)
ELSIF phase >= 2001 AND phase <= 2099 THEN
  idx := phase - 2001;

  IF idx < batch_count THEN
    ui := batch_list[idx + 1];
    STC_CreateTasks(i_unit := ui, io_schedule := g_schedule, io_task := g_task);
    (* phase + 1 → next batch *)
  ELSE
    next_phase := 2100;
  END_IF;

(* ══════════════════════════════════════════════════════════════ *)
(* PHASE 2100: SORT_TASKS                                       *)
(* ══════════════════════════════════════════════════════════════ *)
ELSIF phase = 2100 THEN
  STC_SortTasks(i_trans := 0, i_time_s := i_time_s, io_task := g_task, io_batch := g_batch);
  IF NOT locks_initialized THEN
    lock_cnt := 0;
    FOR bi := 1 TO MAX_LOCKS DO
      locks[bi].Unit := 0;
      locks[bi].Stage := 0;
      locks[bi].Direction := 0;
    END_FOR;
    locks_initialized := TRUE;
  END_IF;
  (* phase + 1 → 2101 *)

(* ══════════════════════════════════════════════════════════════ *)
(* PHASE 2101: SWAP_TASKS                                       *)
(* ══════════════════════════════════════════════════════════════ *)
ELSIF phase = 2101 THEN
  STC_SwapTasks(io_task := g_task);
  (* phase + 1 → 2102 *)

(* ══════════════════════════════════════════════════════════════ *)
(* PHASE 2102: ANALYZE                                          *)
(* ══════════════════════════════════════════════════════════════ *)
ELSIF phase = 2102 THEN
  TSK_Analyze(io_task := g_task,
    o_has_conflict => an_conflict, o_conf_type => an_conf_type,
    o_conf_unit => an_conf_unit, o_conf_stage => an_conf_stage,
    o_conf_trans => an_conf_trans, o_blocked_unit => an_blocked_unit,
    o_blocked_stage => an_blocked_stage, o_deficit => an_deficit);
  o_conflict := an_conflict;

  IF an_conflict THEN
    g_dbg_tsk_conflict_type  := an_conf_type;
    g_dbg_tsk_conf_unit      := an_conf_unit;
    g_dbg_tsk_conf_stage     := an_conf_stage;
    g_dbg_tsk_blocked_unit   := an_blocked_unit;
    g_dbg_tsk_blocked_stage  := an_blocked_stage;
    g_dbg_tsk_deficit        := REAL_TO_DINT(an_deficit);
    g_conflict_resolved := FALSE;
    (* phase + 1 → 2103 RESOLVE *)
  ELSE
    g_conflict_resolved := TRUE;
    next_phase := 2200;   (* skip RESOLVE → NO_TREATMENT *)
  END_IF;

(* ══════════════════════════════════════════════════════════════ *)
(* PHASE 2103: RESOLVE — one conflict, then re-analyze          *)
(* ══════════════════════════════════════════════════════════════ *)
ELSIF phase = 2103 THEN
  TSK_Resolve(
    i_conf_unit     := an_conf_unit,
    i_conf_stage    := an_conf_stage,
    i_conf_trans    := an_conf_trans,
    i_blocked_unit  := an_blocked_unit,
    i_blocked_stage := an_blocked_stage,
    i_deficit       := an_deficit,
    io_locks        := locks,
    io_lock_cnt     := lock_cnt,
    io_schedule     := g_schedule,
    io_task         := g_task,
    io_batch        := g_batch,
    o_total_adv     => rs_total_adv,
    o_total_delay   => rs_total_delay
  );

  (* Collect stretches *)
  IF rs_total_adv > 0.1 AND stretch_cnt < 20 THEN
    stretch_cnt := stretch_cnt + 1;
    stretches[stretch_cnt].Unit   := an_blocked_unit;
    stretches[stretch_cnt].Stage  := an_blocked_stage;
    stretches[stretch_cnt].DelayS := -REAL_TO_DINT(rs_total_adv);
    g_dbg_tsk_total_adv := g_dbg_tsk_total_adv + REAL_TO_DINT(rs_total_adv);
  END_IF;
  IF rs_total_delay > 0.1 AND stretch_cnt < 20 THEN
    stretch_cnt := stretch_cnt + 1;
    stretches[stretch_cnt].Unit   := an_conf_unit;
    stretches[stretch_cnt].Stage  := an_conf_stage;
    stretches[stretch_cnt].DelayS := REAL_TO_DINT(rs_total_delay);
    g_dbg_tsk_total_delay := g_dbg_tsk_total_delay + REAL_TO_DINT(rs_total_delay);
  END_IF;

  conflict_iter := conflict_iter + 1;

  IF conflict_iter >= MAX_CONFLICT_ITER THEN
    g_conflict_resolved := TRUE;
    next_phase := 2200;   (* accept partial, move on *)
  ELSE
    next_phase := 2100;   (* re-SORT → SWAP → ANALYZE *)
  END_IF;

(* ══════════════════════════════════════════════════════════════ *)
(* PHASE 2200: NO_TREATMENT — create no-treatment tasks         *)
(* ══════════════════════════════════════════════════════════════ *)
ELSIF phase = 2200 THEN
  STC_ManualTask(i_time_s := i_time_s, io_task := g_task);
  TSK_NoTreatment(i_time_s := i_time_s, io_task := g_task);
  o_conflict := FALSE;
  (* phase + 1 → 2201 *)

(* ══════════════════════════════════════════════════════════════ *)
(* PHASE 2201: APPLY_STRETCHES — persist resolve decisions      *)
(* ══════════════════════════════════════════════════════════════ *)
ELSIF phase = 2201 THEN
  FOR si := 1 TO stretch_cnt DO
    IF stretches[si].Unit >= 1 AND stretches[si].Unit <= MAX_UNITS THEN
     IF stretches[si].Stage >= 1
        AND stretches[si].Stage <= TreatmentPrograms[stretches[si].Unit].StepCount THEN
      new_cal := TreatmentPrograms[stretches[si].Unit].Steps[stretches[si].Stage].CalTime
               + stretches[si].DelayS;
      IF new_cal < TreatmentPrograms[stretches[si].Unit].Steps[stretches[si].Stage].MinTime THEN
        new_cal := TreatmentPrograms[stretches[si].Unit].Steps[stretches[si].Stage].MinTime;
      END_IF;
      (* Flex cap: min + factor × (max - min) *)
      flex_cap := TreatmentPrograms[stretches[si].Unit].Steps[stretches[si].Stage].MinTime
               + REAL_TO_DINT(SCH_TSK_FLEX_FACTOR * DINT_TO_REAL(
                   TreatmentPrograms[stretches[si].Unit].Steps[stretches[si].Stage].MaxTime
                 - TreatmentPrograms[stretches[si].Unit].Steps[stretches[si].Stage].MinTime));
      IF new_cal > flex_cap THEN
        new_cal := flex_cap;
      END_IF;
      TreatmentPrograms[stretches[si].Unit].Steps[stretches[si].Stage].CalTime := new_cal;

      IF g_batch[stretches[si].Unit].CurStage = stretches[si].Stage THEN
        g_batch[stretches[si].Unit].CalTime := new_cal;
      END_IF;
     END_IF;
    END_IF;
  END_FOR;
  stretch_cnt := 0;
  (* phase + 1 → 2202 *)

(* ══════════════════════════════════════════════════════════════ *)
(* PHASE 2202: MOVE_AWAY — idle transporter move-away check     *)
(* ══════════════════════════════════════════════════════════════ *)
ELSIF phase = 2202 THEN
  STC_TakeOut(i_time_s := i_time_s);
  next_phase := 10000;

(* ══════════════════════════════════════════════════════════════ *)
(* PHASE 10000: READY — cycle complete                          *)
(* ══════════════════════════════════════════════════════════════ *)
ELSIF phase = 10000 THEN
  total_tasks := 0;
  FOR ti := 1 TO MAX_TRANSPORTERS DO
    total_tasks := total_tasks + g_task[ti].Count;
  END_FOR;
  o_task_cnt := total_tasks;

  IF NOT o_conflict THEN
    g_dbg_tsk_conflict_type := 0;
    g_dbg_tsk_conf_unit     := 0;
    g_dbg_tsk_conf_stage    := 0;
    g_dbg_tsk_blocked_unit  := 0;
    g_dbg_tsk_blocked_stage := 0;
    g_dbg_tsk_deficit       := 0;
  END_IF;
  g_dbg_tsk_conflict_iter := conflict_iter;
  g_dbg_tsk_stretch_cnt   := stretch_cnt;

  FOR ui := 1 TO MAX_UNITS DO
    IF g_batch[ui].CurStage >= 1
       AND g_batch[ui].CurStage <= TreatmentPrograms[ui].StepCount THEN
      g_dbg_prog_cal[ui] := TreatmentPrograms[ui].Steps[g_batch[ui].CurStage].CalTime;
    ELSE
      g_dbg_prog_cal[ui] := 0;
    END_IF;
  END_FOR;
  (* phase + 1 → 10001 *)

(* ══════════════════════════════════════════════════════════════ *)
(* PHASE 10001: CHECK_DEP_PENDING                               *)
(* ══════════════════════════════════════════════════════════════ *)
ELSIF phase = 10001 THEN
  IF g_dep_pending.Valid THEN
    FOR ui := 1 TO MAX_UNITS DO
      IF g_dep_pending.Programs[ui].ProgramId > 0 THEN
        TreatmentPrograms[ui] := g_dep_pending.Programs[ui];
      END_IF;
    END_FOR;
    IF g_dep_pending.BatchUnit >= 1 AND g_dep_pending.BatchUnit <= MAX_UNITS THEN
      g_batch[g_dep_pending.BatchUnit].CurStage   := g_dep_pending.BatchStage;
      g_batch[g_dep_pending.BatchUnit].State       := g_dep_pending.BatchState;
      g_batch[g_dep_pending.BatchUnit].StartTime   := g_dep_pending.TimeStamp;
      g_batch[g_dep_pending.BatchUnit].MinTime     := g_dep_pending.BatchMinTime;
      g_batch[g_dep_pending.BatchUnit].MaxTime     := g_dep_pending.BatchMaxTime;
      g_batch[g_dep_pending.BatchUnit].CalTime     := g_dep_pending.BatchCalTime;
    END_IF;
    (* Apply active batch CalTimes written by DEP *)
    FOR ui := 1 TO MAX_UNITS DO
      IF g_dep_pending.ActiveBatchCalTime[ui] > 0
         AND ui <> g_dep_pending.BatchUnit THEN
        g_batch[ui].CalTime := g_dep_pending.ActiveBatchCalTime[ui];
      END_IF;
    END_FOR;
    g_dep_pending.Valid := FALSE;
    g_conflict_resolved := FALSE;
    g_tsk_stable := FALSE;
    next_phase := 1;   (* full recalculation *)
  END_IF;
  (* else phase + 1 → 10002 *)

(* ══════════════════════════════════════════════════════════════ *)
(* PHASE 10002: RESTART — begin new cycle                       *)
(* ══════════════════════════════════════════════════════════════ *)
ELSIF phase = 10002 THEN
  cycle_count := cycle_count + 1;
  o_cycle_cnt := cycle_count;
  o_round_ticks := round_ticks;
  round_ticks := 0;
  next_phase := 1;

(* ══════════════════════════════════════════════════════════════ *)
(* Unknown phase → reset                                        *)
(* ══════════════════════════════════════════════════════════════ *)
ELSE
  next_phase := 1;
END_IF;

(* ── Phase advancement: default = phase + 1 ── *)
IF next_phase > 0 THEN
  phase := next_phase;
ELSE
  phase := phase + 1;
END_IF;
o_phase := phase;

END_FUNCTION_BLOCK

(* ---- TSK_FB_SwapTasks.st ---- *)
(* ============================================================
   TSK_FB_SwapTasks — Swap same-station task pairs
   ============================================================
   Ported from transporterTaskScheduler.js swapSameStationTasks()

   For each transporter queue, checks consecutive task pairs:
   if prev.SinkStationTarget == next.LiftStationTarget AND different units,
   swap order so the lift happens first (avoids deadlock).

   Operates on g_task[1..3] in-place.
   ============================================================ *)

FUNCTION_BLOCK TSK_FB_SwapTasks
VAR_EXTERNAL CONSTANT
    MAX_Transporters : INT;
END_VAR

VAR_EXTERNAL
  g_task : ARRAY[1..MAX_Transporters] OF UDT_JC_TskQueueType;
END_VAR
VAR_OUTPUT
  o_swap_count : INT;   (* number of swaps performed *)
END_VAR
VAR
  ti     : INT;    (* transporter loop *)
  qi     : INT;    (* queue pair index *)
  cnt    : INT;    (* queue count *)
  tmp    : UDT_JC_TskTaskType;  (* swap scratch *)
END_VAR

o_swap_count := 0;

FOR ti := 1 TO MAX_Transporters DO
  cnt := g_task[ti].Count;
  IF cnt >= 2 THEN
    FOR qi := 1 TO cnt - 1 DO
      (* Check: different units AND prev.sink == next.lift *)
      IF g_task[ti].Queue[qi].Unit <> g_task[ti].Queue[qi + 1].Unit
         AND g_task[ti].Queue[qi].SinkStationTarget = g_task[ti].Queue[qi + 1].LiftStationTarget THEN
        (* Swap *)
        tmp := g_task[ti].Queue[qi];
        g_task[ti].Queue[qi] := g_task[ti].Queue[qi + 1];
        g_task[ti].Queue[qi + 1] := tmp;
        o_swap_count := o_swap_count + 1;
      END_IF;
    END_FOR;
  END_IF;
END_FOR;

END_FUNCTION_BLOCK
